// Device/Application/DS6
PROGRAM DS6
VAR
	//massa de dosagem do equipamento em Tonelada.
	MASSA:REAL;
	//Velocidade calculda do Dosador em Hz
	VELOCIDADE:REAL;
	//Espera o fluidizador baixar para o peso minino, pois atingiu o peso maximo
	ESPERA_FLUIDIZADOR_BAIXAR_PESO:BOOL;
	//Liga Dosador manual
	LIGA_DS_MANUAL:BOOL;
	//Liga Dosador automatico
	LIGA_DS_AUTO:BOOL;	
END_VAR

//Dosador 6 - sistema antigo ===============================================
//Formula
//    Passo 1:     massa := (tonelada de dosagem * Percentual de dosagem(sem conversao)  * 10)  
//    Passo 2:    Velocidade := ((massa / (altura * largura * densidade * 60)) + PRST_CONSTANTE_A)/PRST_CONSTANTE_B   	
//	  Inicialmente a Constante a:= 0,045046135
//	  Inicialmente a Constante b:= 0,103503475


//Calculo de velocidade ====================================================

//Calcuulo da massa de dosagem do equipamento 
MASSA := (PRST_VEL_PH1_MANUAL * 10 * PRST_PERC_DOSA_DS06 );

//Calculo da velocidade
VELOCIDADE := ((MASSA/(PRST_ALTURA_DS6*PRST_LARGURA_DS6*PRST_DENSIDADE_DS6*60)) + PRST_CONSTANTE_A_DS6)/PRST_CONSTANTE_B_DS6 ; 

IF BTS_MAPH1 = FALSE THEN
	
	//Comando ==================================================================
	IF BTS_DS6 = TRUE AND AL_GERAL = FALSE THEN
		IF LIGA_DS_MANUAL = TRUE THEN
			LIGA_DS_MANUAL := FALSE;			
		ELSE
			LIGA_DS_MANUAL := TRUE;	
		END_IF		
		BTS_DS6 := FALSE;	
	ELSIF AL_GERAL = TRUE THEN  //delsiga em caso de alarme
		LIGA_DS_MANUAL := FALSE;
		BTS_DS6 := FALSE;	
	END_IF	
	
	//em manual desliga comando do automatico
	LIGA_DS_AUTO := FALSE;
	
ELSE
	
	//Liga dosador 
	IF  AL_GERAL = FALSE THEN
		LIGA_DS_AUTO :=TRUE;
	ELSE
		LIGA_DS_AUTO := FALSE;
	END_IF	
	
	//em auto desliga comando do manual
	LIGA_DS_MANUAL := FALSE;
	
END_IF

//zera velocidade do ph com peso maximo
IF LEITURA_PESO_FLUI1 >= PRST_PESO_MAX_FLUID1 THEN
	ESPERA_FLUIDIZADOR_BAIXAR_PESO := TRUE;
END_IF
	
//ativa velocidade do ph com peso minimo
IF LEITURA_PESO_FLUI1 <= PRST_PESO_MIN_FLUID1 THEN
	ESPERA_FLUIDIZADOR_BAIXAR_PESO := FALSE;
END_IF

IF ESPERA_FLUIDIZADOR_BAIXAR_PESO = FALSE THEN
	//Calculo dosagem kg/h em manual
	PRST_VEL_DS6 := VELOCIDADE;
ELSE
	PRST_VEL_DS6 := 0;
END_IF


//Liga dosador
IF LIGA_DS_AUTO = TRUE OR LIGA_DS_MANUAL = TRUE THEN
	SD_DS6 := TRUE;
ELSE
	SD_DS6 := FALSE;
END_IF

//move velocidade
IF SD_DS6 = TRUE THEN
	VEL_DSA6 :=  PRST_VEL_DS6;
	LEITURA_VEL_DSA6 := PRST_VEL_DS6;
ELSE
	VEL_DSA6 :=0;	
	LEITURA_VEL_DSA6 := 0;
END_IF

END_PROGRAM

// Device/Application/DSA7
PROGRAM DSA7
VAR
	//Tempo de Homogenização em TIME
	TEMPO_DESLIGA_ZERAEVENTO:TON;
	//desliga botao limpa evento
	DESLIGA_BT_LIMPA_EVE:BOOL;
	//Liga Dosador manual
	LIGA_DS_MANUAL:BOOL;
	//Liga Dosador automatico
	LIGA_DS_AUTO:BOOL;
	//Espera o fluidizador baixar para o peso minino, pois atingiu o peso maximo
	ESPERA_FLUIDIZADOR_BAIXAR_PESO:BOOL;
		//Tempo desliga reset totalizador 1
	TMR_RESET_TOTAL1:TON;
	//Tempo desliga reset totalizador 2
	TMR_RESET_TOTAL2:TON;
END_VAR

//POU relacionado aos comandos e alarmes do Dosador Gravimetrico 7 MECHATRON D-5A linha 2


//Controle manual PH 2

//IF BTS_MAPH2 = FALSE THEN
//============================================================================
// comandos manuais 
//============================================================================	
	
//Liga dosador 
IF BTS_DS7 = TRUE AND AL_GERAL = FALSE THEN
	IF LIGA_DS_MANUAL = TRUE THEN
		LIGA_DS_MANUAL := FALSE;
		DS07_HAB := FALSE;
	ELSE
		LIGA_DS_MANUAL :=TRUE;
		DS07_HAB := TRUE;
	END_IF
	BTS_DS7 := FALSE;
END_IF

//desliga em caso de alarme
IF AL_GERAL = TRUE THEN
		LIGA_DS_MANUAL := FALSE;
END_IF

PRST_VEL_DS7 := LEITURA_BASE_SOP_TORRE * (PRST_PERC_DOSA_DS07 / 100);

//============================================================================
// comandos automatico
//============================================================================		
	
//Liga dosador 
IF SD_VLR = TRUE AND SOPRO_SEM_PH = FALSE AND AL_GERAL = FALSE THEN	
	LIGA_DS_AUTO :=TRUE;
	PRST_VEL_DS7 := LEITURA_BASE_SOP_TORRE * (PRST_PERC_DOSA_DS07 / 100);
ELSE
	LIGA_DS_AUTO := FALSE;
	PRST_VEL_DS7 := 0;
END_IF

//Liga dosador
IF LIGA_DS_AUTO = TRUE AND LIGA_DS_MANUAL = TRUE AND AL_GERAL = FALSE THEN
	LIGA_DS7 := TRUE;
	SD_RoscaCelquim := TRUE; 
ELSE
	LIGA_DS7 := FALSE;
	SD_RoscaCelquim := FALSE; 
END_IF


//============================================================================
//  escrita da velocidade
//============================================================================

//Inversão da word da variavel da GVLPH: PRST_VEL_DS7, para variavel da GVLSCHENCK: PESO_DSA7
%QW15080 := %QW12744;
%QW15082 := %QW12742;

//============================================================================
// comandos que independem do comando manual/auto
//============================================================================

//conta tempo de homogenização
TEMPO_DESLIGA_ZERAEVENTO(IN:=BTS_LIMPEVE_DS7,PT:=T#10S);
DESLIGA_BT_LIMPA_EVE := TEMPO_DESLIGA_ZERAEVENTO.Q ;

IF DESLIGA_BT_LIMPA_EVE = TRUE THEN
	BTS_LIMPEVE_DS7 := FALSE;
END_IF

//bits de comando ============================================================
//Os bits de escrita inicio e parada da balança é invertido, por exemplo, para ligar o bit0 = false, e para parar o bit1=false

//Bit iniciar balança
IF LIGA_DS7 = FALSE THEN
	%QX15011.0 := FALSE;    //bit de ligar dosador, false para ativar	
ELSE
	%QX15011.0 := TRUE;		//bit de ligar dosador, true desativa	
END_IF

//bit parar balança
IF LIGA_DS7 = FALSE THEN
	%QX15011.1 := TRUE;		//bit de desligar dosador, true desativar
ELSE		
	%QX15011.1 := FALSE;	//bit de desligar dosador, false ativa	
END_IF

//bit limpar eventos
IF BTS_LIMPEVE_DS7 = TRUE THEN
	%QX15011.2 := TRUE;
ELSE
	%QX15011.2 := FALSE;
END_IF

//bit liberar
%QX15011.3 := TRUE;

//bit modo Volumetrico
IF BTS_MODVOL_DS7 = TRUE THEN
	%QX15011.4 := TRUE;
ELSE
	%QX15011.4 := FALSE;
END_IF
	
//bit modo Gravimetrico
IF BTS_MODGRAV_DS7 = TRUE THEN
	%QX15011.5 := TRUE;
ELSE
	%QX15011.5 := FALSE;
END_IF

//bit reinicializar Totalizador 1
IF BTS_ZERATOTAL1_DS7 = TRUE THEN
	%QX15011.6 := TRUE;
ELSE
	%QX15011.6 := FALSE;
END_IF

//Comando do Reset dos totalizadores geral, apontamento de producao
BTS_ZERATOTAL1_DS7 := BTS_RESET_TOTAL_SCHENCK;
//Tempo desliga reset totalizador 1
TMR_RESET_TOTAL1(IN:= BTS_ZERATOTAL1_DS7, PT:= T#15S);
//desliga o reset do totalizador ao zerar 
IF TMR_RESET_TOTAL1.Q = TRUE THEN
	BTS_ZERATOTAL1_DS7 := FALSE;
	BTS_RESET_TOTAL_SCHENCK := FALSE;
END_IF

//bit reinicializar Totalizador 2
IF BTS_ZERATOTAL2_DS7 = TRUE THEN
	%QX15011.7 := TRUE;
ELSE
	%QX15011.7 := FALSE;
END_IF
//Tempo desliga reset totalizador 2
TMR_RESET_TOTAL2(IN:= BTS_ZERATOTAL2_DS7, PT:= T#15S);
//desliga o reset do totalizador ao zerar 
IF TMR_RESET_TOTAL2.Q = TRUE THEN
	BTS_ZERATOTAL2_DS7 := FALSE;
END_IF


//bit Volume Sincrono
%QX15010.0 := TRUE;

//bit corre. umidade on
%QX15010.1 := TRUE;

//bit corre. umidade off
%QX15010.2 := TRUE;

//bit acionamento med. off
%QX15010.3 := TRUE;

//bit retorno da comporta PMS
%QX15010.4 := TRUE;

//bit reservado
%QX15010.5 := TRUE;

//bit reservado
%QX15010.6 := TRUE;

//bit reservado
%QX15010.7 := TRUE;


//====================================================================================
// Leitura Valores REAL 
//====================================================================================

//Totalizador1, leitura em Kg, 
//Inversão da word da variavel da GVLSCHENCK: LEITURA_TOTALIZADOR1_DSA7, para variavel da GVLPH: TOTALIZADOR1_KG 
%QW10080 := %IW15152;
%QW10082 := %IW15150;

//Totalizador2, leitura em Kg, apenas invertidos as words
//Inversão da word da variavel da GVLSCHENCK: LEITURA_TOTALIZADOR2_DSA7, para variavel da GVLPH: TOTALIZADOR2_KG 
%QW10084 := %IW15212;
%QW10086 := %IW15210;

//Totalizador3, leitura em Tonelada, invertidos as words e dividido por 1000 
//Inversão da word da variavel da GVLSCHENCK: LEITURA_TOTALIZADOR3_DSA7, para variavel da GVLPH: TOTALIZADOR3_KG 
%QW10088 := %IW15322;
%QW10090 := %IW15320;
TOTALIZADOR3_TON_DS7 := TOTALIZADOR3_KG_DS7 / 1000;

//Velocidade atual do dosador
%QW10320 := %IW15272;
%QW10322 := %IW15270;

VELOCIDADE_REAL_DS7 := VELOCIDADE_REAL2_DS7 ;

END_PROGRAM

// Device/Application/DSA8
PROGRAM DSA8
VAR
	//Tempo de Homogenização em TIME
	TEMPO_DESLIGA_ZERAEVENTO:TON;
	//desliga botao limpa evento
	DESLIGA_BT_LIMPA_EVE:BOOL;
	//Liga Dosador manual
	LIGA_DS_MANUAL:BOOL;
	//Liga Dosador automatico
	LIGA_DS_AUTO:BOOL;
	//Espera o fluidizador baixar para o peso minino, pois atingiu o peso maximo
	ESPERA_FLUIDIZADOR_BAIXAR_PESO:BOOL;
	//Tempo desliga reset totalizador 1
	TMR_RESET_TOTAL1:TON;
	//Tempo desliga reset totalizador 2
	TMR_RESET_TOTAL2:TON;
END_VAR

//POU relacionado aos comandos e alarmes do Dosador Gravimetrico 8 MECHATRON D-7A linha 2


//Controle manual PH 2

IF BTS_MAPH2 = FALSE THEN
//============================================================================
// comandos manuais 
//============================================================================	
	
	//Liga dosador 
	IF BTS_DS8 = TRUE AND AL_GERAL = FALSE THEN
		IF LIGA_DS_MANUAL = TRUE THEN
			LIGA_DS_MANUAL := FALSE;
		ELSE
			LIGA_DS_MANUAL :=TRUE;
		END_IF
		BTS_DS8 := FALSE;
	END_IF
	//desliga em caso de alarme
	IF AL_GERAL = TRUE THEN
		LIGA_DS_MANUAL := FALSE;
	END_IF

	//Calculo dosagem kg/h em manual
	PRST_VEL_DS8 := (PRST_VEL_PH2_MANUAL * 1000) * (PRST_PERC_DOSA_DS08 / 100);
	
	//em manual desliga comando do automatico
	LIGA_DS_AUTO := FALSE;	
ELSE
	
//============================================================================
// comandos automatico
//============================================================================		
	
	//Liga dosador 
	IF  AL_GERAL = FALSE THEN
		LIGA_DS_AUTO :=TRUE;
	ELSE
		LIGA_DS_AUTO := FALSE;
	END_IF
	
	//zera velocidade do ph com peso maximo
	IF LEITURA_PESO_FLUI2 >= PRST_PESO_MAX_FLUID2 THEN
		ESPERA_FLUIDIZADOR_BAIXAR_PESO := TRUE;
	END_IF
	
	//ativa velocidade do ph com peso minimo
	IF LEITURA_PESO_FLUI2 <= PRST_PESO_MIN_FLUID2 THEN
		ESPERA_FLUIDIZADOR_BAIXAR_PESO := FALSE;
	END_IF
	
	IF ESPERA_FLUIDIZADOR_BAIXAR_PESO = FALSE THEN
		//Calculo dosagem kg/h em manual
		PRST_VEL_DS8 := (VELOCIDADE_PH2_AUTO) * (PRST_PERC_DOSA_DS08 / 100);
	ELSE
		PRST_VEL_DS8 := 0;
	END_IF
	
	
	//em auto desliga comando do manual
	LIGA_DS_MANUAL := FALSE;
END_IF

//Liga dosador
IF LIGA_DS_AUTO = TRUE OR LIGA_DS_MANUAL = TRUE THEN
	LIGA_DS8 := TRUE;
ELSE
	LIGA_DS8 := FALSE;
END_IF

//============================================================================
//  escrita da velocidade
//============================================================================

//Inversão da word da variavel da GVLPH: PRST_VEL_DS8, para variavel da GVLSCHENCK: PESO_DSA8
%QW15084 := %QW12748;
%QW15086 := %QW12746;

//============================================================================
// comandos que independem do comando manual/auto
//============================================================================

//conta tempo de homogenização
TEMPO_DESLIGA_ZERAEVENTO(IN:=BTS_LIMPEVE_DS8,PT:=T#10S);
DESLIGA_BT_LIMPA_EVE := TEMPO_DESLIGA_ZERAEVENTO.Q ;

IF DESLIGA_BT_LIMPA_EVE = TRUE THEN
	BTS_LIMPEVE_DS8 := FALSE;
END_IF

//bits de comando ============================================================
//Os bits de escrita inicio e parada da balança é invertido, por exemplo, para ligar o bit0 = false, e para parar o bit1=false

//Bit iniciar balança
IF LIGA_DS8 = FALSE THEN
	%QX15013.0 := FALSE;    //bit de ligar dosador, false para ativar	
ELSE
	%QX15013.0 := TRUE;		//bit de ligar dosador, true desativa	
END_IF

//bit parar balança
IF LIGA_DS8 = FALSE THEN
	%QX15013.1 := TRUE;		//bit de desligar dosador, true desativar
ELSE		
	%QX15013.1 := FALSE;	//bit de desligar dosador, false ativa	
END_IF

//bit limpar eventos
IF BTS_LIMPEVE_DS8 = TRUE THEN
	%QX15013.2 := TRUE;
ELSE
	%QX15013.2 := FALSE;
END_IF

//bit liberar
%QX15013.3 := TRUE;

//bit modo Volumetrico
IF BTS_MODVOL_DS8 = TRUE THEN
	%QX15013.4 := TRUE;
ELSE
	%QX15013.4 := FALSE;
END_IF
	
//bit modo Gravimetrico
IF BTS_MODGRAV_DS8 = TRUE THEN
	%QX15013.5 := TRUE;
ELSE
	%QX15013.5 := FALSE;
END_IF

//bit reinicializar Totalizador 1
IF BTS_ZERATOTAL1_DS8 = TRUE THEN
	%QX15013.6 := TRUE;
ELSE
	%QX15013.6 := FALSE;
END_IF

//Comando do Reset dos totalizadores geral, apontamento de producao
BTS_ZERATOTAL1_DS8 := BTS_RESET_TOTAL_SCHENCK;
//Tempo desliga reset totalizador 1
TMR_RESET_TOTAL1(IN:= BTS_ZERATOTAL1_DS8, PT:= T#15S);
//desliga o reset do totalizador ao zerar 
IF TMR_RESET_TOTAL1.Q = TRUE THEN
	BTS_ZERATOTAL1_DS8 := FALSE;
	BTS_RESET_TOTAL_SCHENCK := FALSE;
END_IF

//bit reinicializar Totalizador 2
IF BTS_ZERATOTAL2_DS8 = TRUE THEN
	%QX15013.7 := TRUE;
ELSE
	%QX15013.7 := FALSE;
END_IF
//Tempo desliga reset totalizador 2
TMR_RESET_TOTAL2(IN:= BTS_ZERATOTAL2_DS8, PT:= T#15S);
//desliga o reset do totalizador ao zerar 
IF TMR_RESET_TOTAL2.Q = TRUE THEN
	BTS_ZERATOTAL2_DS8 := FALSE;
END_IF

//bit Volume Sincrono
%QX15012.0 := TRUE;

//bit corre. umidade on
%QX15012.1 := TRUE;

//bit corre. umidade off
%QX15012.2 := TRUE;

//bit acionamento med. off
%QX15012.3 := TRUE;

//bit retorno da comporta PMS
%QX15012.4 := TRUE;

//bit reservado
%QX15012.5 := TRUE;

//bit reservado
%QX15012.6 := TRUE;

//bit reservado
%QX15012.7 := TRUE;


//====================================================================================
// Leitura Valores REAL 
//====================================================================================

//Totalizador1, leitura em Kg, 
//Inversão da word da variavel da GVLSCHENCK: LEITURA_TOTALIZADOR1_DSA8, para variavel da GVLPH: TOTALIZADOR1_KG 
%QW10096 := %IW15156;
%QW10098 := %IW15154;

//Totalizador2, leitura em Kg, apenas invertidos as words
//Inversão da word da variavel da GVLSCHENCK: LEITURA_TOTALIZADOR2_DSA8, para variavel da GVLPH: TOTALIZADOR2_KG 
%QW10100 := %IW15216;
%QW10102 := %IW15214;

//Totalizador3, leitura em Tonelada, invertidos as words e dividido por 1000 
//Inversão da word da variavel da GVLSCHENCK: LEITURA_TOTALIZADOR3_DSA8, para variavel da GVLPH: TOTALIZADOR3_KG 
%QW10104 := %IW15326;
%QW10106 := %IW15324;
TOTALIZADOR3_TON_DS8 := TOTALIZADOR3_KG_DS8 / 1000;

//Velocidade atual do dosador
%QW10324 := %IW15276;
%QW10326 := %IW15274;

VELOCIDADE_REAL_DS8 := VELOCIDADE_REAL2_DS8 ;

END_PROGRAM

// Device/Application/DSA9
PROGRAM DSA9
VAR
	//Tempo de Homogenização em TIME
	TEMPO_DESLIGA_ZERAEVENTO:TON;
	//desliga botao limpa evento
	DESLIGA_BT_LIMPA_EVE:BOOL;
	//Liga Dosador manual
	LIGA_DS_MANUAL:BOOL;
	//Liga Dosador automatico
	LIGA_DS_AUTO:BOOL;
	//Espera o fluidizador baixar para o peso minino, pois atingiu o peso maximo
	ESPERA_FLUIDIZADOR_BAIXAR_PESO:BOOL;
	//Tempo desliga reset totalizador 1
	TMR_RESET_TOTAL1:TON;
	//Tempo desliga reset totalizador 2
	TMR_RESET_TOTAL2:TON;

END_VAR

//POU relacionado aos comandos e alarmes do Dosador Gravimetrico 9 MECHATRON D-6A linha 2	


//Controle manual PH 2

IF BTS_MAPH2 = FALSE THEN
//============================================================================
// comandos manuais 
//============================================================================	
	
	//Liga dosador 
	IF BTS_DS9 = TRUE AND AL_GERAL = FALSE THEN
		IF LIGA_DS_MANUAL = TRUE THEN
			LIGA_DS_MANUAL := FALSE;
		ELSE
			LIGA_DS_MANUAL :=TRUE;
		END_IF
		BTS_DS9 := FALSE;
	END_IF
	//desliga em caso de alarme
	IF AL_GERAL = TRUE THEN
		LIGA_DS_MANUAL := FALSE;
	END_IF
	
	//Calculo dosagem kg/h em manual
	PRST_VEL_DS9 := (PRST_VEL_PH2_MANUAL * 1000) * (PRST_PERC_DOSA_DS09 / 100);

	//em manual desliga comando do automatico
	LIGA_DS_AUTO := FALSE;
	
ELSE
	
//============================================================================
// comandos automatico
//============================================================================		
	
	//Liga dosador 
	IF  AL_GERAL = FALSE THEN
		LIGA_DS_AUTO :=TRUE;
	ELSE
		LIGA_DS_AUTO := FALSE;
	END_IF
	
	//zera velocidade do ph com peso maximo
	IF LEITURA_PESO_FLUI2 >= PRST_PESO_MAX_FLUID2 THEN
		ESPERA_FLUIDIZADOR_BAIXAR_PESO := TRUE;
	END_IF
	
	//ativa velocidade do ph com peso minimo
	IF LEITURA_PESO_FLUI2 <= PRST_PESO_MIN_FLUID2 THEN
		ESPERA_FLUIDIZADOR_BAIXAR_PESO := FALSE;
	END_IF
	
	IF ESPERA_FLUIDIZADOR_BAIXAR_PESO = FALSE THEN
		//Calculo dosagem kg/h em manual
		PRST_VEL_DS9 := (VELOCIDADE_PH2_AUTO) * (PRST_PERC_DOSA_DS09 / 100);
	ELSE
		PRST_VEL_DS9 := 0;	
	END_IF
	
	
	//em auto desliga comando do manual
	LIGA_DS_MANUAL := FALSE;
END_IF

//Liga dosador
IF LIGA_DS_AUTO = TRUE OR LIGA_DS_MANUAL = TRUE THEN
	LIGA_DS9 := TRUE;
ELSE
	LIGA_DS9 := FALSE;
END_IF

//============================================================================
//  escrita da velocidade
//============================================================================

//Inversão da word da variavel da GVLPH: PRST_VEL_DS9, para variavel da GVLSCHENCK: PESO_DSA9
%QW15088 := %QW12752;
%QW15090 := %QW12750;


//============================================================================
// comandos que independem do comando manual/auto
//============================================================================

//conta tempo de homogenização
TEMPO_DESLIGA_ZERAEVENTO(IN:=BTS_LIMPEVE_DS9,PT:=T#10S);
DESLIGA_BT_LIMPA_EVE := TEMPO_DESLIGA_ZERAEVENTO.Q ;

IF DESLIGA_BT_LIMPA_EVE = TRUE THEN
	BTS_LIMPEVE_DS9 := FALSE;
END_IF

//bits de comando ============================================================
//Os bits de escrita inicio e parada da balança é invertido, por exemplo, para ligar o bit0 = false, e para parar o bit1=false

//Bit iniciar balança
IF LIGA_DS9 = FALSE THEN
	%QX15015.0 := FALSE;    //bit de ligar dosador, false para ativar	
ELSE
	%QX15015.0 := TRUE;		//bit de ligar dosador, true desativa	
END_IF

//bit parar balança
IF LIGA_DS9 = FALSE THEN
	%QX15015.1 := TRUE;		//bit de desligar dosador, true desativar
ELSE		
	%QX15015.1 := FALSE;	//bit de desligar dosador, false ativa	
END_IF

//bit limpar eventos
IF BTS_LIMPEVE_DS9 = TRUE THEN
	%QX15015.2 := TRUE;
ELSE
	%QX15015.2 := FALSE;
END_IF

//bit liberar
%QX15015.3 := TRUE;

//bit modo Volumetrico
IF BTS_MODVOL_DS9 = TRUE THEN
	%QX15015.4 := TRUE;
ELSE
	%QX15015.4 := FALSE;
END_IF
	
//bit modo Gravimetrico
IF BTS_MODGRAV_DS9 = TRUE THEN
	%QX15015.5 := TRUE;
ELSE
	%QX15015.5 := FALSE;
END_IF

//bit reinicializar Totalizador 1
IF BTS_ZERATOTAL1_DS9 = TRUE THEN
	%QX15015.6 := TRUE;
ELSE
	%QX15015.6 := FALSE;
END_IF

//Comando do Reset dos totalizadores geral, apontamento de producao
BTS_ZERATOTAL1_DS9 := BTS_RESET_TOTAL_SCHENCK;
//Tempo desliga reset totalizador 1
TMR_RESET_TOTAL1(IN:= BTS_ZERATOTAL1_DS9, PT:= T#15S);
//desliga o reset do totalizador ao zerar 
IF TMR_RESET_TOTAL1.Q = TRUE THEN
	BTS_ZERATOTAL1_DS9 := FALSE;
	BTS_RESET_TOTAL_SCHENCK := FALSE;
END_IF

//bit reinicializar Totalizador 2
IF BTS_ZERATOTAL2_DS9 = TRUE THEN
	%QX15015.7 := TRUE;
ELSE
	%QX15015.7 := FALSE;
END_IF
//Tempo desliga reset totalizador 2
TMR_RESET_TOTAL2(IN:= BTS_ZERATOTAL2_DS9, PT:= T#15S);
//desliga o reset do totalizador ao zerar 
IF TMR_RESET_TOTAL2.Q = TRUE THEN
	BTS_ZERATOTAL2_DS9 := FALSE;
END_IF

//bit Volume Sincrono
%QX15014.0 := TRUE;

//bit corre. umidade on
%QX15014.1 := TRUE;

//bit corre. umidade off
%QX15014.2 := TRUE;

//bit acionamento med. off
%QX15014.3 := TRUE;

//bit retorno da comporta PMS
%QX15014.4 := TRUE;

//bit reservado
%QX15014.5 := TRUE;

//bit reservado
%QX15014.6 := TRUE;

//bit reservado
%QX15014.7 := TRUE;


//====================================================================================
// Leitura Valores REAL 
//====================================================================================

//Totalizador1, leitura em Kg, 
//Inversão da word da variavel da GVLSCHENCK: LEITURA_TOTALIZADOR1_DSA9, para variavel da GVLPH: TOTALIZADOR1_KG 
%QW10112 := %IW15160;
%QW10114 := %IW15158;

//Totalizador2, leitura em Kg, apenas invertidos as words
//Inversão da word da variavel da GVLSCHENCK: LEITURA_TOTALIZADOR2_DSA9, para variavel da GVLPH: TOTALIZADOR2_KG 
%QW10116 := %IW15220;
%QW10118 := %IW15218;

//Totalizador3, leitura em Tonelada, invertidos as words e dividido por 1000 
//Inversão da word da variavel da GVLSCHENCK: LEITURA_TOTALIZADOR3_DSA9, para variavel da GVLPH: TOTALIZADOR3_KG 
%QW10120 := %IW15330;
%QW10122 := %IW15328;
TOTALIZADOR3_TON_DS9 := TOTALIZADOR3_KG_DS9 / 1000;

//Velocidade atual do dosador
%QW10328 := %IW15280;
%QW10330 := %IW15278;

VELOCIDADE_REAL_DS9 := VELOCIDADE_REAL2_DS9;

END_PROGRAM

// Device/Application/DSA10
PROGRAM DSA10
VAR
	//Tempo de Homogenização em TIME
	TEMPO_DESLIGA_ZERAEVENTO:TON;
	//desliga botao limpa evento
	DESLIGA_BT_LIMPA_EVE:BOOL;
	//Liga Dosador manual
	LIGA_DS_MANUAL:BOOL;
	//Liga Dosador automatico
	LIGA_DS_AUTO:BOOL;
	//Espera o fluidizador baixar para o peso minino, pois atingiu o peso maximo
	ESPERA_FLUIDIZADOR_BAIXAR_PESO:BOOL;
	//Tempo desliga reset totalizador 1
	TMR_RESET_TOTAL1:TON;
	//Tempo desliga reset totalizador 2
	TMR_RESET_TOTAL2:TON;
END_VAR

//POU relacionado aos comandos e alarmes do Dosador Gravimetrico 10 MECHATRON DEA-4A linha 2	


//Controle manual PH 2

IF BTS_MAPH2 = FALSE THEN
//============================================================================
// comandos manuais 
//============================================================================	
	
	//Liga dosador 
	IF BTS_DS10 = TRUE AND AL_GERAL = FALSE THEN
		IF LIGA_DS_MANUAL = TRUE THEN
			LIGA_DS_MANUAL := FALSE;
		ELSE
			LIGA_DS_MANUAL :=TRUE;
		END_IF
		BTS_DS10 := FALSE;
	END_IF
	//desliga em caso de alarme
	IF AL_GERAL = TRUE THEN
		LIGA_DS_MANUAL := FALSE;
	END_IF

	//Calculo dosagem kg/h em manual
	PRST_VEL_DS10 := (PRST_VEL_PH2_MANUAL * 1000) * (PRST_PERC_DOSA_DS10 / 100);
	
	
	//em manual desliga comando do automatico
	LIGA_DS_AUTO := FALSE;
	
ELSE
//============================================================================
// comandos automatico
//============================================================================		
	
	//Liga dosador 
	IF  AL_GERAL = FALSE THEN
		LIGA_DS_AUTO :=TRUE;
	ELSE
		LIGA_DS_AUTO := FALSE;
	END_IF
	
	
	//zera velocidade do ph com peso maximo
	IF LEITURA_PESO_FLUI2 >= PRST_PESO_MAX_FLUID2 THEN
		ESPERA_FLUIDIZADOR_BAIXAR_PESO := TRUE;
	END_IF
	
	//ativa velocidade do ph com peso minimo
	IF LEITURA_PESO_FLUI2 <= PRST_PESO_MIN_FLUID2 THEN
		ESPERA_FLUIDIZADOR_BAIXAR_PESO := FALSE;
	END_IF
	
	IF ESPERA_FLUIDIZADOR_BAIXAR_PESO = FALSE THEN
		//Calculo dosagem kg/h em manual
		PRST_VEL_DS10 := (VELOCIDADE_PH2_AUTO) * (PRST_PERC_DOSA_DS10 / 100);
	ELSE
		PRST_VEL_DS10 := 0;
	END_IF
	
	//em auto desliga comando do manual
	LIGA_DS_MANUAL := FALSE;
	
END_IF

//Liga dosador
IF LIGA_DS_AUTO = TRUE OR LIGA_DS_MANUAL = TRUE THEN
	LIGA_DS10 := TRUE;
ELSE
	LIGA_DS10 := FALSE;
END_IF

//============================================================================
//  escrita da velocidade
//============================================================================

//Inversão da word da variavel da GVLPH: PRST_VEL_DS10, para variavel da GVLSCHENCK: PESO_DSA10
%QW15092 := %QW12756;
%QW15094 := %QW12754;

//============================================================================
// comandos que independem do comando manual/auto
//============================================================================

//conta tempo de homogenização
TEMPO_DESLIGA_ZERAEVENTO(IN:=BTS_LIMPEVE_DS10,PT:=T#10S);
DESLIGA_BT_LIMPA_EVE := TEMPO_DESLIGA_ZERAEVENTO.Q ;

IF DESLIGA_BT_LIMPA_EVE = TRUE THEN
	BTS_LIMPEVE_DS10 := FALSE;
END_IF

//bits de comando ============================================================
//Os bits de escrita inicio e parada da balança é invertido, por exemplo, para ligar o bit0 = false, e para parar o bit1=false

//Bit iniciar balança
IF LIGA_DS10 = FALSE THEN
	%QX15017.0 := FALSE;    //bit de ligar dosador, false para ativar	
ELSE
	%QX15017.0 := TRUE;		//bit de ligar dosador, true desativa	
END_IF

//bit parar balança
IF LIGA_DS10 = FALSE THEN
	%QX15017.1 := TRUE;		//bit de desligar dosador, true desativar
ELSE		
	%QX15017.1 := FALSE;	//bit de desligar dosador, false ativa	
END_IF

//bit limpar eventos
IF BTS_LIMPEVE_DS10 = TRUE THEN
	%QX15017.2 := TRUE;
ELSE
	%QX15017.2 := FALSE;
END_IF

//bit liberar
%QX15017.3 := TRUE;

//bit modo Volumetrico
IF BTS_MODVOL_DS10 = TRUE THEN
	%QX15017.4 := TRUE;
ELSE
	%QX15017.4 := FALSE;
END_IF
	
//bit modo Gravimetrico
IF BTS_MODGRAV_DS10 = TRUE THEN
	%QX15017.5 := TRUE;
ELSE
	%QX15017.5 := FALSE;
END_IF

//bit reinicializar Totalizador 1
IF BTS_ZERATOTAL1_DS10 = TRUE THEN
	%QX15017.6 := TRUE;
ELSE
	%QX15017.6 := FALSE;
END_IF

//Comando do Reset dos totalizadores geral, apontamento de producao
BTS_ZERATOTAL1_DS10 := BTS_RESET_TOTAL_SCHENCK;
//Tempo desliga reset totalizador 1
TMR_RESET_TOTAL1(IN:= BTS_ZERATOTAL1_DS10, PT:= T#15S);
//desliga o reset do totalizador ao zerar 
IF TMR_RESET_TOTAL1.Q = TRUE THEN
	BTS_ZERATOTAL1_DS10 := FALSE;
	BTS_RESET_TOTAL_SCHENCK := FALSE;
END_IF

//bit reinicializar Totalizador 2
IF BTS_ZERATOTAL2_DS10 = TRUE THEN
	%QX15017.7 := TRUE;
ELSE
	%QX15017.7 := FALSE;
END_IF
//Tempo desliga reset totalizador 2
TMR_RESET_TOTAL2(IN:= BTS_ZERATOTAL2_DS10, PT:= T#15S);
//desliga o reset do totalizador ao zerar 
IF TMR_RESET_TOTAL2.Q = TRUE THEN
	BTS_ZERATOTAL2_DS10 := FALSE;
END_IF

//bit Volume Sincrono
%QX15016.0 := TRUE;

//bit corre. umidade on
%QX15016.1 := TRUE;

//bit corre. umidade off
%QX15016.2 := TRUE;

//bit acionamento med. off
%QX15016.3 := TRUE;

//bit retorno da comporta PMS
%QX15016.4 := TRUE;

//bit reservado
%QX15016.5 := TRUE;

//bit reservado
%QX15016.6 := TRUE;

//bit reservado
%QX15016.7 := TRUE;


//====================================================================================
// Leitura Valores REAL 
//====================================================================================

//Totalizador1, leitura em Kg, 
//Inversão da word da variavel da GVLSCHENCK: LEITURA_TOTALIZADOR1_DSA10, para variavel da GVLPH: TOTALIZADOR1_KG 
%QW10128 := %IW15164;
%QW10130 := %IW15162;

//Totalizador2, leitura em Kg, apenas invertidos as words
//Inversão da word da variavel da GVLSCHENCK: LEITURA_TOTALIZADOR2_DSA10, para variavel da GVLPH: TOTALIZADOR2_KG 
%QW10132 := %IW15224;
%QW10134 := %IW15222;

//Totalizador3, leitura em Tonelada, invertidos as words e dividido por 1000 
//Inversão da word da variavel da GVLSCHENCK: LEITURA_TOTALIZADOR3_DSA10, para variavel da GVLPH: TOTALIZADOR3_KG 
%QW10136 := %IW15334;
%QW10138 := %IW15332;
TOTALIZADOR3_TON_DS10 := TOTALIZADOR3_KG_DS10 / 1000;

//Velocidade atual do dosador
%QW10332 := %IW15284;
%QW10334 := %IW15282;

VELOCIDADE_REAL_DS10 := VELOCIDADE_REAL2_DS10;

END_PROGRAM

// Device/Application/DSA11
PROGRAM DSA11
VAR
	//Tempo de Homogenização em TIME
	TEMPO_DESLIGA_ZERAEVENTO:TON;
	//desliga botao limpa evento
	DESLIGA_BT_LIMPA_EVE:BOOL;
	//Liga Dosador manual
	LIGA_DS_MANUAL:BOOL;
	//Liga Dosador automatico
	LIGA_DS_AUTO:BOOL; 
	//Espera o fluidizador baixar para o peso minino, pois atingiu o peso maximo
	ESPERA_FLUIDIZADOR_BAIXAR_PESO:BOOL;
	//Tempo desliga reset totalizador 1
	TMR_RESET_TOTAL1:TON;
	//Tempo desliga reset totalizador 2
	TMR_RESET_TOTAL2:TON;
END_VAR

//POU relacionado aos comandos e alarmes do Dosador Gravimetrico 11 MECHATRON DEA-2A linha 2 - Po Base 11


//Controle manual PH 2

IF BTS_MAPH2 = FALSE THEN
//============================================================================
// comandos manuais 
//============================================================================	
	
	//Liga dosador 
	IF BTS_DS11 = TRUE AND AL_GERAL = FALSE THEN
		IF LIGA_DS_MANUAL = TRUE THEN
			LIGA_DS_MANUAL := FALSE;
		ELSE
			LIGA_DS_MANUAL :=TRUE;
		END_IF
		BTS_DS11 := FALSE;
	END_IF
	//desliga em caso de alarme
	IF AL_GERAL = TRUE THEN
		LIGA_DS_MANUAL := FALSE;
	END_IF
	
	//Calculo dosagem kg/h em manual
	PRST_VEL_DS11 := (PRST_VEL_PH2_MANUAL * 1000) * (PRST_PERC_DOSA_PB11 / 100);		
	
	//em manual desliga comando do automatico
	LIGA_DS_AUTO := FALSE;
	
ELSE
//============================================================================
// comandos automatico
//============================================================================		
	
	//Liga dosador 
	IF  AL_GERAL = FALSE THEN
		LIGA_DS_AUTO :=TRUE;
	ELSE
		LIGA_DS_AUTO := FALSE;
	END_IF
	
	//zera velocidade do ph com peso maximo
	IF LEITURA_PESO_FLUI2 >= PRST_PESO_MAX_FLUID2 THEN
		ESPERA_FLUIDIZADOR_BAIXAR_PESO := TRUE;
	END_IF
	
	//ativa velocidade do ph com peso minimo
	IF LEITURA_PESO_FLUI2 <= PRST_PESO_MIN_FLUID2 THEN
		ESPERA_FLUIDIZADOR_BAIXAR_PESO := FALSE;
	END_IF

	IF ESPERA_FLUIDIZADOR_BAIXAR_PESO = FALSE THEN
		//Calculo dosagem kg/h em manual
		PRST_VEL_DS11 := (VELOCIDADE_PH2_AUTO) * (PRST_PERC_DOSA_PB11 / 100);
	ELSE
		PRST_VEL_DS11 := 0;
	END_IF
	
	
	//em auto desliga comando do manual
	LIGA_DS_MANUAL := FALSE;
	
END_IF

//Liga dosador
IF LIGA_DS_AUTO = TRUE OR LIGA_DS_MANUAL = TRUE THEN
	LIGA_DS11 := TRUE;
ELSE
	LIGA_DS11 := FALSE;
END_IF


//============================================================================
//  escrita da velocidade
//============================================================================

//Inversão da word da variavel da GVLPH: PRST_VEL_DS11, para variavel da GVLSCHENCK: PESO_DSA11
%QW15096 := %QW12760;
%QW15098 := %QW12758;

//============================================================================
// comandos que independem do comando manual/auto
//============================================================================

//conta tempo de homogenização
TEMPO_DESLIGA_ZERAEVENTO(IN:=BTS_LIMPEVE_DS11,PT:=T#10S);
DESLIGA_BT_LIMPA_EVE := TEMPO_DESLIGA_ZERAEVENTO.Q ;

IF DESLIGA_BT_LIMPA_EVE = TRUE THEN
	BTS_LIMPEVE_DS11 := FALSE;
END_IF

//bits de comando ============================================================
//Os bits de escrita inicio e parada da balança é invertido, por exemplo, para ligar o bit0 = false, e para parar o bit1=false

//Bit iniciar balança
IF LIGA_DS11 = FALSE THEN
	%QX15019.0 := FALSE;    //bit de ligar dosador, false para ativar	
ELSE
	%QX15019.0 := TRUE;		//bit de ligar dosador, true desativa	
END_IF

//bit parar balança
IF LIGA_DS11 = FALSE THEN
	%QX15019.1 := TRUE;		//bit de desligar dosador, true desativar
ELSE		
	%QX15019.1 := FALSE;	//bit de desligar dosador, false ativa	
END_IF

//bit limpar eventos
IF BTS_LIMPEVE_DS11 = TRUE THEN
	%QX15019.2 := TRUE;
ELSE
	%QX15019.2 := FALSE;
END_IF

//bit liberar
%QX15019.3 := TRUE;

//bit modo Volumetrico
IF BTS_MODVOL_DS11 = TRUE THEN
	%QX15019.4 := TRUE;
ELSE
	%QX15019.4 := FALSE;
END_IF
	
//bit modo Gravimetrico
IF BTS_MODGRAV_DS11 = TRUE THEN
	%QX15019.5 := TRUE;
ELSE
	%QX15019.5 := FALSE;
END_IF

//bit reinicializar Totalizador 1
IF BTS_ZERATOTAL1_DS11 = TRUE THEN
	%QX15019.6 := TRUE;
ELSE
	%QX15019.6 := FALSE;
END_IF

//Comando do Reset dos totalizadores geral, apontamento de producao
BTS_ZERATOTAL1_DS11 := BTS_RESET_TOTAL_SCHENCK;
//Tempo desliga reset totalizador 1
TMR_RESET_TOTAL1(IN:= BTS_ZERATOTAL1_DS11, PT:= T#15S);
//desliga o reset do totalizador ao zerar 
IF TMR_RESET_TOTAL1.Q = TRUE THEN
	BTS_ZERATOTAL1_DS11 := FALSE;
	BTS_RESET_TOTAL_SCHENCK := FALSE;
END_IF

//bit reinicializar Totalizador 2
IF BTS_ZERATOTAL2_DS11 = TRUE THEN
	%QX15019.7 := TRUE;
ELSE
	%QX15019.7 := FALSE;
END_IF
//Tempo desliga reset totalizador 2
TMR_RESET_TOTAL2(IN:= BTS_ZERATOTAL2_DS11, PT:= T#15S);
//desliga o reset do totalizador ao zerar 
IF TMR_RESET_TOTAL2.Q = TRUE THEN
	BTS_ZERATOTAL2_DS11 := FALSE;
END_IF

//bit Volume Sincrono
%QX15018.0 := TRUE;

//bit corre. umidade on
%QX15018.1 := TRUE;

//bit corre. umidade off
%QX15018.2 := TRUE;

//bit acionamento med. off
%QX15018.3 := TRUE;

//bit retorno da comporta PMS
%QX15018.4 := TRUE;

//bit reservado
%QX15018.5 := TRUE;

//bit reservado
%QX15018.6 := TRUE;

//bit reservado
%QX15018.7 := TRUE;


//====================================================================================
// Leitura Valores REAL 
//====================================================================================

//Totalizador1, leitura em Kg, 
//Inversão da word da variavel da GVLSCHENCK: LEITURA_TOTALIZADOR1_DSA11, para variavel da GVLPH: TOTALIZADOR1_KG 
%QW10144 := %IW15168;
%QW10146 := %IW15166;

//Totalizador2, leitura em Kg, apenas invertidos as words
//Inversão da word da variavel da GVLSCHENCK: LEITURA_TOTALIZADOR2_DSA11, para variavel da GVLPH: TOTALIZADOR2_KG 
%QW10148 := %IW15228;
%QW10150 := %IW15226;

//Totalizador3, leitura em Tonelada, invertidos as words e dividido por 1000 
//Inversão da word da variavel da GVLSCHENCK: LEITURA_TOTALIZADOR3_DSA11, para variavel da GVLPH: TOTALIZADOR3_KG 
%QW10152 := %IW15338;
%QW10154 := %IW15336;
TOTALIZADOR3_TON_DS11 := TOTALIZADOR3_KG_DS11 / 1000;

//Velocidade atual do dosador
%QW10336 := %IW15288;
%QW10338 := %IW15286;

VELOCIDADE_REAL_DS11 := VELOCIDADE_REAL2_DS11;

END_PROGRAM

// Device/Application/DSA12
PROGRAM DSA12
VAR
	//Tempo de Homogenização em TIME
	TEMPO_DESLIGA_ZERAEVENTO:TON;
	//desliga botao limpa evento
	DESLIGA_BT_LIMPA_EVE:BOOL;
	//Liga Dosador manual
	LIGA_DS_MANUAL:BOOL;
	//Liga Dosador automatico
	LIGA_DS_AUTO:BOOL;
	//Espera o fluidizador baixar para o peso minino, pois atingiu o peso maximo
	ESPERA_FLUIDIZADOR_BAIXAR_PESO:BOOL;
	//Tempo desliga reset totalizador 1
	TMR_RESET_TOTAL1:TON;
	//Tempo desliga reset totalizador 2
	TMR_RESET_TOTAL2:TON;
END_VAR

//POU relacionado aos comandos e alarmes do Dosador Gravimetrico 12 MECHATRON DEA-3A linha 2	


//Controle manual PH 2

IF BTS_MAPH2 = FALSE THEN
//============================================================================
// comandos manuais 
//============================================================================	
	
	//Liga dosador 
	IF BTS_DS12 = TRUE AND AL_GERAL = FALSE THEN
		IF LIGA_DS_MANUAL = TRUE THEN
			LIGA_DS_MANUAL := FALSE;
		ELSE
			LIGA_DS_MANUAL :=TRUE;
		END_IF
		BTS_DS12 := FALSE;
	END_IF
	//desliga em caso de alarme
	IF AL_GERAL = TRUE THEN
		LIGA_DS_MANUAL := FALSE;
	END_IF

	//Calculo dosagem kg/h em manual
	PRST_VEL_DS12 := (PRST_VEL_PH2_MANUAL * 1000) * (PRST_PERC_DOSA_DS12 / 100);
	
	//em manual desliga comando do automatico
	LIGA_DS_AUTO := FALSE;	
ELSE
//============================================================================
// comandos automatico
//============================================================================		
	
	//Liga dosador 
	IF  AL_GERAL = FALSE THEN
		LIGA_DS_AUTO :=TRUE;
	ELSE
		LIGA_DS_AUTO := FALSE;
	END_IF
	
	//zera velocidade do ph com peso maximo
	IF LEITURA_PESO_FLUI2 >= PRST_PESO_MAX_FLUID2 THEN
		ESPERA_FLUIDIZADOR_BAIXAR_PESO := TRUE;
	END_IF
	
	//ativa velocidade do ph com peso minimo
	IF LEITURA_PESO_FLUI2 <= PRST_PESO_MIN_FLUID2 THEN
		ESPERA_FLUIDIZADOR_BAIXAR_PESO := FALSE;
	END_IF
	
	IF ESPERA_FLUIDIZADOR_BAIXAR_PESO = FALSE THEN
		//Calculo dosagem kg/h em manual
		PRST_VEL_DS12 := (VELOCIDADE_PH2_AUTO) * (PRST_PERC_DOSA_DS12 / 100);
	ELSE
		PRST_VEL_DS12 := 0;
	END_IF
	
	//em auto desliga comando do manual
	LIGA_DS_MANUAL := FALSE;
	
END_IF

//Liga dosador
IF LIGA_DS_AUTO = TRUE OR LIGA_DS_MANUAL = TRUE THEN
	LIGA_DS12 := TRUE;
ELSE
	LIGA_DS12 := FALSE;
END_IF

//============================================================================
//  escrita da velocidade
//============================================================================

//Inversão da word da variavel da GVLPH: PRST_VEL_DS12, para variavel da GVLSCHENCK: PESO_DSA12
%QW15100 := %QW12764;
%QW15102 := %QW12762;

//============================================================================
// comandos que independem do comando manual/auto
//============================================================================

//conta tempo de homogenização
TEMPO_DESLIGA_ZERAEVENTO(IN:=BTS_LIMPEVE_DS12,PT:=T#10S);
DESLIGA_BT_LIMPA_EVE := TEMPO_DESLIGA_ZERAEVENTO.Q ;

IF DESLIGA_BT_LIMPA_EVE = TRUE THEN
	BTS_LIMPEVE_DS12 := FALSE;
END_IF

//bits de comando ============================================================
//Os bits de escrita inicio e parada da balança é invertido, por exemplo, para ligar o bit0 = false, e para parar o bit1=false

//Bit iniciar balança
IF LIGA_DS12 = FALSE THEN
	%QX15021.0 := FALSE;    //bit de ligar dosador, false para ativar	
ELSE
	%QX15021.0 := TRUE;		//bit de ligar dosador, true desativa	
END_IF

//bit parar balança
IF LIGA_DS12 = FALSE THEN
	%QX15021.1 := TRUE;		//bit de desligar dosador, true desativar
ELSE		
	%QX15021.1 := FALSE;	//bit de desligar dosador, false ativa	
END_IF

//bit limpar eventos
IF BTS_LIMPEVE_DS12 = TRUE THEN
	%QX15021.2 := TRUE;
ELSE
	%QX15021.2 := FALSE;
END_IF

//bit liberar
%QX15021.3 := TRUE;

//bit modo Volumetrico
IF BTS_MODVOL_DS12 = TRUE THEN
	%QX15021.4 := TRUE;
ELSE
	%QX15021.4 := FALSE;
END_IF
	
//bit modo Gravimetrico
IF BTS_MODGRAV_DS12 = TRUE THEN
	%QX15021.5 := TRUE;
ELSE
	%QX15021.5 := FALSE;
END_IF

//bit reinicializar Totalizador 1
IF BTS_ZERATOTAL1_DS12 = TRUE THEN
	%QX15021.6 := TRUE;
ELSE
	%QX15021.6 := FALSE;
END_IF

//Comando do Reset dos totalizadores geral, apontamento de producao
BTS_ZERATOTAL1_DS12 := BTS_RESET_TOTAL_SCHENCK;
//Tempo desliga reset totalizador 1
TMR_RESET_TOTAL1(IN:= BTS_ZERATOTAL1_DS12, PT:= T#15S);
//desliga o reset do totalizador ao zerar 
IF TMR_RESET_TOTAL1.Q = TRUE THEN
	BTS_ZERATOTAL1_DS12 := FALSE;
	BTS_RESET_TOTAL_SCHENCK := FALSE;
END_IF

//bit reinicializar Totalizador 2
IF BTS_ZERATOTAL2_DS12 = TRUE THEN
	%QX15021.7 := TRUE;
ELSE
	%QX15021.7 := FALSE;
END_IF
//Tempo desliga reset totalizador 2
TMR_RESET_TOTAL2(IN:= BTS_ZERATOTAL2_DS12, PT:= T#15S);
//desliga o reset do totalizador ao zerar 
IF TMR_RESET_TOTAL2.Q = TRUE THEN
	BTS_ZERATOTAL2_DS12 := FALSE;
END_IF

//bit Volume Sincrono
%QX15020.0 := TRUE;

//bit corre. umidade on
%QX15020.1 := TRUE;

//bit corre. umidade off
%QX15020.2 := TRUE;

//bit acionamento med. off
%QX15020.3 := TRUE;

//bit retorno da comporta PMS
%QX15020.4 := TRUE;

//bit reservado
%QX15020.5 := TRUE;

//bit reservado
%QX15020.6 := TRUE;

//bit reservado
%QX15020.7 := TRUE;


//====================================================================================
// Leitura Valores REAL 
//====================================================================================

//Totalizador1, leitura em Kg, 
//Inversão da word da variavel da GVLSCHENCK: LEITURA_TOTALIZADOR1_DSA12, para variavel da GVLPH: TOTALIZADOR1_KG 
%QW10160 := %IW15172;
%QW10162 := %IW15170;

//Totalizador2, leitura em Kg, apenas invertidos as words
//Inversão da word da variavel da GVLSCHENCK: LEITURA_TOTALIZADOR2_DSA12, para variavel da GVLPH: TOTALIZADOR2_KG 
%QW10164 := %IW15232;
%QW10166 := %IW15230;

//Totalizador3, leitura em Tonelada, invertidos as words e dividido por 1000 
//Inversão da word da variavel da GVLSCHENCK: LEITURA_TOTALIZADOR3_DSA12, para variavel da GVLPH: TOTALIZADOR3_KG 
%QW10168 := %IW15342;
%QW10170 := %IW15340;
TOTALIZADOR3_TON_DS12 := TOTALIZADOR3_KG_DS12 / 1000;

//Velocidade atual do dosador
%QW10340 := %IW15292;
%QW10342 := %IW15290;

VELOCIDADE_REAL_DS12 := VELOCIDADE_REAL2_DS12;

END_PROGRAM

// Device/Application/DSA14
PROGRAM DSA14
VAR
	//Tempo de Homogenização em TIME
	TEMPO_DESLIGA_ZERAEVENTO:TON;
	//desliga botao limpa evento
	DESLIGA_BT_LIMPA_EVE:BOOL;
	//Liga Dosador manual
	LIGA_DS_MANUAL:BOOL;
	//Liga Dosador automatico
	LIGA_DS_AUTO:BOOL;
	//Espera o fluidizador baixar para o peso minino, pois atingiu o peso maximo
	ESPERA_FLUIDIZADOR_BAIXAR_PESO:BOOL;
	//Tempo desliga reset totalizador 1
	TMR_RESET_TOTAL1:TON;
	//Tempo desliga reset totalizador 2
	TMR_RESET_TOTAL2:TON;
	teste1: WORD;
	teste2: WORD;
	teste3: DWORD;
END_VAR

//POU relacionado aos comandos e alarmes do Dosador Gravimetrico 14 MECHATRON DEA-3A linha 2	


//Controle manual PH 2

IF BTS_MAPH2 = FALSE THEN
//============================================================================
// comandos manuais 
//============================================================================	
	
	//Liga dosador 
	IF BTS_DS14 = TRUE AND AL_GERAL = FALSE THEN
		IF LIGA_DS_MANUAL = TRUE THEN
			LIGA_DS_MANUAL := FALSE;
		ELSE
			LIGA_DS_MANUAL :=TRUE;
		END_IF
		BTS_DS14 := FALSE;
	END_IF
	//desliga em caso de alarme
	IF AL_GERAL = TRUE THEN
		LIGA_DS_MANUAL := FALSE;
	END_IF

	//Calculo dosagem kg/h em manual
	PRST_VEL_DS14 := (PRST_VEL_PH2_MANUAL * 1000) * (PRST_PERC_DOSA_DS14 / 100);
	
	//em manual desliga comando do automatico
	LIGA_DS_AUTO := FALSE;	
ELSE
//============================================================================
// comandos automatico
//============================================================================		
	
	//Liga dosador 
	IF  AL_GERAL = FALSE THEN
		LIGA_DS_AUTO :=TRUE;
	ELSE
		LIGA_DS_AUTO := FALSE;
	END_IF
	
	//zera velocidade do ph com peso maximo
	IF LEITURA_PESO_FLUI2 >= PRST_PESO_MAX_FLUID2 THEN
		ESPERA_FLUIDIZADOR_BAIXAR_PESO := TRUE;
	END_IF
	
	//ativa velocidade do ph com peso minimo
	IF LEITURA_PESO_FLUI2 <= PRST_PESO_MIN_FLUID2 THEN
		ESPERA_FLUIDIZADOR_BAIXAR_PESO := FALSE;
	END_IF
	
	IF ESPERA_FLUIDIZADOR_BAIXAR_PESO = FALSE THEN
		//Calculo dosagem kg/h em manual
		PRST_VEL_DS14 := (VELOCIDADE_PH2_AUTO) * (PRST_PERC_DOSA_DS14 / 100);
	ELSE
		PRST_VEL_DS14 := 0;
	END_IF
	
	//em auto desliga comando do manual
	LIGA_DS_MANUAL := FALSE;
	
END_IF

//Liga dosador
IF (( LIGA_DS_AUTO = TRUE  OR LIGA_DS_MANUAL = TRUE) ) THEN
	LIGA_DS14 := TRUE;
ELSE
	LIGA_DS14 := FALSE;
END_IF

//============================================================================
//  escrita da velocidade
//============================================================================

//Inversão da word da variavel da GVLPH: PRST_VEL_DS14, para variavel da GVLSCHENCK: PESO_DSA14
%QW15108 := %QW13578; // Endereço 852
%QW15110 := %QW13576; // Endereço 851




//============================================================================
// comandos que independem do comando manual/auto
//============================================================================

//conta tempo de homogenização
TEMPO_DESLIGA_ZERAEVENTO(IN:=BTS_LIMPEVE_DS14,PT:=T#10S);
DESLIGA_BT_LIMPA_EVE := TEMPO_DESLIGA_ZERAEVENTO.Q ;

IF DESLIGA_BT_LIMPA_EVE = TRUE THEN
	BTS_LIMPEVE_DS14 := FALSE;
END_IF

//bits de comando ============================================================
//Os bits de escrita inicio e parada da balança é invertido, por exemplo, para ligar o bit0 = false, e para parar o bit1=false

//Bit iniciar balança
IF LIGA_DS14 = FALSE THEN
	%QX15025.0 := FALSE;    //bit de ligar dosador, false para ativar	
ELSE
	%QX15025.0 := TRUE;		//bit de ligar dosador, true desativa	
END_IF

//bit parar balança
IF LIGA_DS14 = FALSE THEN
	%QX15025.1 := TRUE;		//bit de desligar dosador, true desativar
ELSE		
	%QX15025.1 := FALSE;	//bit de desligar dosador, false ativa	
END_IF

//bit limpar eventos
IF BTS_LIMPEVE_DS14 = TRUE THEN
	%QX15025.2 := TRUE;
ELSE
	%QX15025.2 := FALSE;
END_IF

//bit liberar
%QX15025.3 := TRUE;

//bit modo Volumetrico
IF BTS_MODVOL_DS14 = TRUE THEN
	%QX15025.4 := TRUE;
ELSE
	%QX15025.4 := FALSE;
END_IF
	
//bit modo Gravimetrico
IF BTS_MODGRAV_DS14 = TRUE THEN
	%QX15025.5 := TRUE;
ELSE
	%QX15025.5 := FALSE;
END_IF

//bit reinicializar Totalizador 1
IF BTS_ZERATOTAL1_DS14 = TRUE THEN
	%QX15025.6 := TRUE;
ELSE
	%QX15025.6 := FALSE;
END_IF

//Comando do Reset dos totalizadores geral, apontamento de producao
BTS_ZERATOTAL1_DS14 := BTS_RESET_TOTAL_SCHENCK;
//Tempo desliga reset totalizador 1
TMR_RESET_TOTAL1(IN:= BTS_ZERATOTAL1_DS14, PT:= T#30S);
//desliga o reset do totalizador ao zerar 
IF TMR_RESET_TOTAL1.Q = TRUE THEN
	BTS_ZERATOTAL1_DS14 := FALSE;
	BTS_RESET_TOTAL_SCHENCK := FALSE;
END_IF

//bit reinicializar Totalizador 2
IF BTS_ZERATOTAL2_DS14 = TRUE THEN
	%QX15025.7 := TRUE;
ELSE
	%QX15025.7 := FALSE;
END_IF
//Tempo desliga reset totalizador 2
TMR_RESET_TOTAL2(IN:= BTS_ZERATOTAL2_DS14, PT:= T#30S);
//desliga o reset do totalizador ao zerar 
IF TMR_RESET_TOTAL2.Q = TRUE THEN
	BTS_ZERATOTAL2_DS14 := FALSE;
END_IF

//bit Volume Sincrono
%QX15024.0 := TRUE;

//bit corre. umidade on
%QX15024.1 := TRUE;

//bit corre. umidade off
%QX15024.2 := TRUE;

//bit acionamento med. off
%QX15024.3 := TRUE;

//bit retorno da comporta PMS
%QX15024.4 := TRUE;

//bit reservado
%QX15024.5 := TRUE;

//bit reservado
%QX15024.6 := TRUE;

//bit reservado
%QX15024.7 := TRUE;


//====================================================================================
// Leitura Valores REAL 
//====================================================================================

//Totalizador1, leitura em Kg, 
//Inversão da word da variavel da GVLSCHENCK: LEITURA_TOTALIZADOR1_DSA14, para variavel da GVLPH: TOTALIZADOR1_KG 
%QW10800 := %IW16304; // Endereço Modbus 1700
%QW10802 := %IW16302; // Endereço Modbus 1701

//Totalizador2, leitura em Kg, apenas invertidos as words
//Inversão da word da variavel da GVLSCHENCK: LEITURA_TOTALIZADOR2_DSA14, para variavel da GVLPH: TOTALIZADOR2_KG 
%QW10804 := %IW16308; // Endereço Modbus 1702
%QW10806 := %IW16306; // Endereço Modbus 1703

//Totalizador3, leitura em Tonelada, invertidos as words e dividido por 1000 
//Inversão da word da variavel da GVLSCHENCK: LEITURA_TOTALIZADOR3_DSA12, para variavel da GVLPH: TOTALIZADOR3_KG 
%QW10808 := %IW16312; // Endereço Modbus 1704
%QW10810 := %IW16310; // Endereço Modbus 1705
TOTALIZADOR3_TON_DS14 := TOTALIZADOR3_KG_DS14 / 1000;

//Velocidade atual do dosador
%QW10848 := %IW16300; // Endereço Modbus 1720
%QW10850 := %IW16298; // Endereço Modbus 1721

VELOCIDADE_REAL_DS14 := VELOCIDADE_REAL2_DS14;

END_PROGRAM

// Device/Application/DSATorre
PROGRAM DSATorre
VAR
	//Rotação das bombas de alta 
	RPM:REAL;
	//P - Volume base incorporada;
	P:REAL;
	PERCENTUAL_BASE:REAL;		
	//Ds  - densidade do slurry em %
	ds:REAL;
	//Us  - Umidade do Slurry em %
	Us:REAL;
	//Ub  - Umidade do po base em %
	Ub:REAL;
	//Velocidade do Dosador
	Q:REAL;	
	//Tempo de Homogenização em TIME
	TEMPO_DESLIGA_ZERAEVENTO:TON;
	//desliga botao limpa evento
	DESLIGA_BT_LIMPA_EVE:BOOL;
	//Liga Dosador manual
	LIGA_DS_MANUAL:BOOL;
	//Liga Dosador automatico
	LIGA_DS_AUTO:BOOL;
	//Tempo desliga reset totalizador 1
	TMR_RESET_TOTAL1:TON;
	//Tempo desliga reset totalizador 2
	TMR_RESET_TOTAL2:TON;
		//Tempo retardo para ligar dosador
	TMR_RETARDO_LIGA_DOSDOR:TON;
	//Liga dosador apos tempo de retardo
	LIGA_DOSADOR_APOS_RETARDO:BOOL;
	//Tempo retardo para mover velocidade para dosador
	TMR_RETARDO_MOVE_VEL_DOSDOR:TON;
	//Move velocidade para dosador
	MOVE_VEL_DOSADOR:BOOL;
END_VAR

//POU relacionado aos comandos e alarmes do Dosador TORRE	MECHATRON DEA-D1
//Formula
//  Se Baseia no calculo de Q considerando as variaveis:
//    - vazão do po base que esta sendo soprado
//    - percental de slfato que se deseja incorporar base
//
//  Q = P*(%base) / % Sulfato
//  
//   P - Volume base incorporada;
//   %base - fraçao de base desejada
//   %sulfato - fraçao sulfato desejado na mistura
//
//    Passo 1:    calculo % base
//					% Base = %Sulfato - 100%
//				
//    Passo 2:     calculo P
//                            P:= ((RPM/11,2)*0,965 * ds * (1 - Us))/ (1 -  Ub)
//
//     RPM - rotacao motor da bomba de alta
//     Ds  - densidade do slurry em gr/l
//     Us  - Umidade do Slurry em %
//     Ub  - Umidade do po base em %
//
//     Passo3: calculo Q
//                             Q = P*PRST_RELACAO_PO_BASE / 100
//  
// multiplicar por 60 no final, pois a velocidade esta em rpm 


//Calculo da velocidade =====================================================

//se apenas bomba de alta 1 ligada
IF SD_BA1 = TRUE AND SD_BA2 = FALSE THEN
	RPM := LEITURA_VEL_ALT1;
ELSIF SD_BA2 = TRUE AND SD_BA1 = FALSE THEN    //se apenas bomba de alta 2 ligada
	RPM := LEITURA_VEL_ALT2;
ELSIF SD_BA2 = TRUE AND SD_BA1 = TRUE THEN
	RPM := LEITURA_VEL_ALT1 + LEITURA_VEL_ALT2;   // se as duas estiverem ligadas
ELSE                //quando nenhuma ligada
	RPM := 0;
END_IF


//calculo P

//Passo 1: 
//            % Base = %Sulfato - 100%

PERCENTUAL_BASE := 100 - PRST_PERC_SULFATO_DSTORRE;


//Passo 2:
//     RPM - rotacao motor da bomba de alta
//     Ds  - densidade do slurry em %
//     Us  - Umidade do Slurry em %
//     Ub  - Umidade do po base em %

ds := PRST_DS_DSTORRE/1000 ; 
Us := PRST_US_DSTORRE/100 ;
Ub := PRST_UB_DSTORRE/100 ;

 P := (((RPM/11.2)*0.965 * ds * (1 - Us))/ (1 -  Ub))*60;

 //Copia informação do P para Supervisório
 LEITURA_BASE_SOP_TORRE := P;
 
 //Passo 3:
//Calculo Q

Q := P*PRST_RELACAO_PO_BASE / 100;


//Retardo para mover velocidade dosador
TMR_RETARDO_MOVE_VEL_DOSDOR(IN:= SD_VLR, PT:= T#10S);
//move velocidade
MOVE_VEL_DOSADOR := TMR_RETARDO_MOVE_VEL_DOSDOR.Q;


//Se não estiver soprando zera velocidade do dosador
IF MOVE_VEL_DOSADOR = TRUE THEN
	PRST_VEL_DSTORRE := Q;
ELSE
	PRST_VEL_DSTORRE := 0;
END_IF



//Liga dosador manualmente ================================
IF BTS_DSTORRE = TRUE AND AL_GERAL = FALSE THEN
	IF LIGA_DS_MANUAL = TRUE THEN
		LIGA_DS_MANUAL := FALSE;
	ELSE
		LIGA_DS_MANUAL :=TRUE;
	END_IF
	BTS_DSTORRE := FALSE;
END_IF
//desliga em caso de alarme
IF AL_GERAL = TRUE THEN
	LIGA_DS_MANUAL := FALSE;
END_IF
//informa que dosador esta habilitado
IF LIGA_DS_MANUAL THEN
	DSATORRE_HAB := TRUE;
ELSE
	DSATORRE_HAB := FALSE;
END_IF

//liga se valvula retorno para torre e sopro com PH	==========================
IF SD_VLR = TRUE AND SOPRO_SEM_PH = FALSE AND AL_GERAL = FALSE THEN	
	LIGA_DS_AUTO :=TRUE;
ELSE
	LIGA_DS_AUTO := FALSE;
END_IF	
		

//Liga dosador
IF LIGA_DS_AUTO = TRUE AND LIGA_DS_MANUAL = TRUE AND AL_GERAL = FALSE  THEN
	LIGA_DSTORRE := TRUE;
ELSE
	LIGA_DSTORRE := FALSE;
END_IF


//Retardo para ligar dosador
TMR_RETARDO_LIGA_DOSDOR(IN:= LIGA_DSTORRE, PT:= T#10S);
//liga dosador
LIGA_DOSADOR_APOS_RETARDO := TMR_RETARDO_LIGA_DOSDOR.Q;

//============================================================================
//  escrita da velocidade
//============================================================================

//Inversão da word da variavel da GVLPH: PRST_VEL_DSTORRE, para variavel da GVLSCHENCK: PESO_DSATORRE
%QW15104 := %QW12768;
%QW15106 := %QW12766;

//============================================================================
// comandos que independem do comando manual/auto
//============================================================================


//bits de comando ============================================================
//Os bits de escrita inicio e parada da balança é invertido, por exemplo, para ligar o bit0 = false, e para parar o bit1=false

//Bit iniciar balança
IF LIGA_DOSADOR_APOS_RETARDO = FALSE THEN
	%QX15023.0 := FALSE;    //bit de ligar dosador, false para ativar	
ELSE
	%QX15023.0 := TRUE;		//bit de ligar dosador, true desativa	
END_IF

//bit parar balança
IF LIGA_DOSADOR_APOS_RETARDO = FALSE THEN
	%QX15023.1 := TRUE;		//bit de desligar dosador, true desativar
ELSE		
	%QX15023.1 := FALSE;	//bit de desligar dosador, false ativa	
END_IF

//bit limpar eventos
IF BTS_LIMPEVE_DSTORRE = TRUE THEN
	%QX15023.2 := TRUE;
ELSE
	%QX15023.2 := FALSE;
END_IF
//===============================RESET LIMPA EVENTOS======================

TEMPO_DESLIGA_ZERAEVENTO(IN:=BTS_LIMPEVE_DSTORRE,PT:=T#3S);
DESLIGA_BT_LIMPA_EVE := TEMPO_DESLIGA_ZERAEVENTO.Q ;

IF DESLIGA_BT_LIMPA_EVE = TRUE THEN
	BTS_LIMPEVE_DSTORRE := FALSE;
END_IF

//===============================RESET LIMPA EVENTOS======================

//bit liberar
%QX15023.3 := TRUE;

//bit modo Volumetrico
IF BTS_MODVOL_DSTORRE = TRUE THEN
	%QX15023.4 := TRUE;
ELSE
	%QX15023.4 := FALSE;
END_IF
	
//bit modo Gravimetrico
IF BTS_MODGRAV_DSTORRE = TRUE THEN
	%QX15023.5 := TRUE;
ELSE
	%QX15023.5 := FALSE;
END_IF

//bit reinicializar Totalizador 1
IF BTS_ZERATOTAL1_DSTORRE = TRUE THEN
	%QX15023.6 := TRUE;
ELSE
	%QX15023.6 := FALSE;
END_IF

//Comando do Reset dos totalizadores geral, apontamento de producao
BTS_ZERATOTAL1_DSTORRE := BTS_RESET_TOTAL_SCHENCK;
//Tempo desliga reset totalizador 1
TMR_RESET_TOTAL1(IN:= BTS_ZERATOTAL1_DSTORRE, PT:= T#15S);
//desliga o reset do totalizador ao zerar 
IF TMR_RESET_TOTAL1.Q = TRUE THEN
	BTS_ZERATOTAL1_DSTORRE := FALSE;
	BTS_RESET_TOTAL_SCHENCK := FALSE;
END_IF

//bit reinicializar Totalizador 2
IF BTS_ZERATOTAL2_DSTORRE = TRUE THEN
	%QX15023.7 := TRUE;
ELSE
	%QX15023.7 := FALSE;
END_IF
//Tempo desliga reset totalizador 2
TMR_RESET_TOTAL2(IN:= BTS_ZERATOTAL2_DSTORRE, PT:= T#15S);
//desliga o reset do totalizador ao zerar 
IF TMR_RESET_TOTAL2.Q = TRUE THEN
	BTS_ZERATOTAL2_DSTORRE := FALSE;
END_IF

//bit Volume Sincrono
%QX15022.0 := TRUE;

//bit corre. umidade on
%QX15022.1 := TRUE;

//bit corre. umidade off
%QX15022.2 := TRUE;

//bit acionamento med. off
%QX15022.3 := TRUE;

//bit retorno da comporta PMS
%QX15022.4 := TRUE;

//bit reservado
%QX15022.5 := TRUE;

//bit reservado
%QX15022.6 := TRUE;

//bit reservado
%QX15022.7 := TRUE;



//====================================================================================
// Leitura Valores REAL 
//====================================================================================

//Totalizador1, leitura em Kg, 
//Inversão da word da variavel da GVLSCHENCK: LEITURA_TOTALIZADOR1_DSATORRE, para variavel da GVLPH: TOTALIZADOR1_KG 
%QW10176 := %IW15176;
%QW10178 := %IW15174;

//Totalizador2, leitura em Kg, apenas invertidos as words
//Inversão da word da variavel da GVLSCHENCK: LEITURA_TOTALIZADOR2_DSATORRE, para variavel da GVLPH: TOTALIZADOR2_KG 
%QW10180 := %IW15236;
%QW10182 := %IW15234;

//Totalizador3, leitura em Tonelada, invertidos as words e dividido por 1000 
//Inversão da word da variavel da GVLSCHENCK: LEITURA_TOTALIZADOR3_DSATORRE, para variavel da GVLPH: TOTALIZADOR3_KG 
%QW10184 := %IW15346;
%QW10186 := %IW15344;
TOTALIZADOR3_TON_DSTORRE := TOTALIZADOR3_KG_DSTORRE / 1000;

//Velocidade atual do dosador
%QW10344 := %IW15296;
%QW10346 := %IW15294;

VELOCIDADE_REAL_DSTORRE := VELOCIDADE_REAL2_DSTORRE ;

END_PROGRAM

// Device/Application/ProdL1
PROGRAM ProdL1
VAR
	//PRODUÇÃO LINHAS ENVASE
	
//=========================	
PULSO_CNT_L1_1T: R_TRIG;
PULSO_CNT_L1_2T: R_TRIG;
PULSO_CNT_L1_3T: R_TRIG;
	CNT_PRD_L1: INT;
	//CNT_L1: BOOL;
//=========================	
	Result : RTC_STATUS;
	DATEANDTIME : EXTENDED_DATE_AND_TIME;
	xEnable : BOOL;
//=========================		
	dia: INT;
	mes: INT;
	ano: INT;
	hora: INT;
	minuto: INT;
	segundo: INT;
	
	
	
	//HoraInicio1Turno: INT;
	//MinInicio1Turno: INT;
	HoraFim1Turno: INT;
	MinFim1Turno: INT;
	//HoraInicio2Turno: INT;
	//MinInicio2Turno: INT;
	HoraFim2Turno: INT;
	MinFim2Turno: INT;
	//HoraInicio3Turno: INT;
	//MinInicio3Turno: INT;
	HoraFim3Turno: INT;
	MinFim3Turno: INT;
	EficienciaL1: INT;
	
	
	HabContL1_1T: BOOL;
	HabContL1_2T: BOOL;
	HabContL1_3T: BOOL;
	
	CNT_PRD_L1_2T: INT;
	CNT_PRD_L1_3T: INT;
	EficienciaL1_1T: REAL;
	EficienciaL1_2T: REAL;
	EficienciaL1_3T: REAL;
	
	MinDispL1_1T: REAL;
	
	ProdL1_1T_realtime: REAL;
	MinDispL1_2T: REAL;
	ProdL1_2T_realtime: REAL;
	EficL1_2T_realtime: REAL;
	MinDispL1_3T: REAL;
	ProdL1_3T_realtime: REAL;
	EficL1_3T_realtime: REAL;
	
	//TMR_SIMUL_CNT1: TON;
	//LIBERA_TMR_SIMUL: BOOL;
	EficL1_2T_projetada: REAL;
	//TMR_SIMUL_CNT2: TON;
	//LIBERA_TMR_SIMUL2T: BOOL;
	//TMR_SIMUL_CNT3: TON;
	//LIBERA_TMR_SIMUL3T: BOOL;
	EficL1_3T_projetada: REAL;
//	EficL1_1T_realtime: REAL;
	HabTemParadaL1: BOOL;
	TempParadaL1: Ton;
	horaParadaL1: INT;
	MinParadaL1: INT;
	RegistraHora: BOOL;
	Borda_des_RegistraHora: F_TRIG;
	HoraRetornoParadaL1: INT;
	MinRetornoParadaL1: INT;
	TempoParadaL1: INT;
	TotalMinParado: TON;
	HabTotalMinParado: BOOL;
	//TempoProduzindo: REAL;
	//MinDispTurnoAtual: REAL;

	refeicao: BOOL;
	DDS: BOOL;
	SETUP: BOOL;
	L1semprogramacao: BOOL;
	
END_VAR


//LÓGICA PARA ANÁLISES DE PRODUTIVADADE DA L1 DE CARTUCHOS
	dia := BYTE_TO_INT (DATEANDTIME.byDayOfMonth);
	mes := BYTE_TO_INT (DATEANDTIME.byMonth);
	ano := WORD_TO_INT (DATEANDTIME.wYear);
	hora := BYTE_TO_INT (DATEANDTIME.byHours);
	minuto := BYTE_TO_INT (DATEANDTIME.byMinutes);
	segundo := BYTE_TO_INT (DATEANDTIME.bySeconds);
	xEnable := TRUE;
	
	//HABILITA RTC==========================
	IF xEnable = TRUE THEN
	Result := GetDateAndTime(DATEANDTIME);
	END_IF
//HABILITA RTC==========================

//=====================1º TURNO ========================
	
		//HoraInicio1Turno: INT;
	
	HoraFim1Turno:= HoraInicio2Turno;
	MinFim1Turno:= MinInicio2Turno;
	HoraFim2Turno:= HoraInicio3Turno;
	MinFim2Turno:= MinInicio3Turno;
	
	//10 minutos - Reunião / DSS / Treinamento
	//20 minutosPartida de linha / Parada de Linha xxxxxxxxxx
	//15 minutosRefeições (Café / Almoço / Janta)xxxxxxxxxxxx
	//60 minutosRefeições (Café / Almoço / Janta)
	//10 minutosPartida de linha / Parada de Linha xxxxxxxxxxxxxx
			
	MinDispL1_1T := (((INT_TO_REAL (HoraFim1Turno) - INT_TO_REAL(HoraInicio1Turno) )*60)-
		INT_TO_REAL(MinInicio1Turno)+INT_TO_REAL(MinFim1Turno)-60-10);
		
			IF TempoProduzindo < 1 THEN
			TempoProduzindo :=0;
		END_IF
	
		//LÓGICA PARA VERIFICAR SE EXISTE ATRASO DE PRODUÇÃO NO INSTANTE ATUAL
		
	IF  CXS_ATRASOL1 >= 0AND HabContL1_1T = TRUE THEN 
	CXS_ATRASOL1:= REAL_TO_INT(ProdL1_1T_realtime)-CNT_PRD_L1_1T;
	END_IF
	IF  CXS_ATRASOL1 >= 0 AND HabContL1_2T = TRUE THEN 
	CXS_ATRASOL1:= REAL_TO_INT(ProdL1_2T_realtime)-CNT_PRD_L1_1T;
	END_IF
	IF  CXS_ATRASOL1 >= 0 AND HabContL1_3T = TRUE THEN 
	CXS_ATRASOL1:=REAL_TO_INT(ProdL1_2T_realtime)-CNT_PRD_L1_1T;
	END_IF
		IF  CXS_ATRASOL1  < 0 THEN 
		CXS_ATRASOL1:= 0;
		END_IF
	
	//LÓGICA PARA VERIFICAR SE EXISTE ATRASO DE PRODUÇÃO NO INSTANTE ATUAL
		
		//LÓGICA PARA CONTAR TEMPO DE PARADA
		TempParadaL1(IN:=HabTemParadaL1 ,PT:= T#30S);
		IF TempParadaL1.Q   THEN
		TotalMinParado(IN:=HabTotalMinParado ,PT:= T#1M);
		IF TotalMinParado.Q = TRUE THEN
			TempoParada := TempoParada+1;
			HabTotalMinParado := FALSE;
			ELSE
				HabTotalMinParado := TRUE;
			END_IF
		END_IF
		
		IF PULSO_CNT_L1_1T.Q = FALSE AND PULSO_CNT_L1_2T.Q = FALSE AND PULSO_CNT_L1_3T.Q = FALSE  THEN
		HabTemParadaL1 := TRUE;
		
		ELSE 	
		HabTemParadaL1 := FALSE;
		END_IF
		//LÓGICA PARA CONTAR TEMPO DE PARADA
//==============Habilita contadores 1º turno ================
IF (hora = HoraInicio1Turno AND minuto = MinInicio1Turno)  THEN
HabContL1_1T := TRUE;
HabContL1_3T := FALSE;
HabContL1_2T := FALSE;
CNT_PRD_L1_3T := 0;
CNT_PRD_L1_2T := 0;
CNT_PRD_L1_1T := 0;
TempoProduzindo :=0;
EficL1_1T_projetada:=0;
EficL1_1T_realtime :=0;
ProdL1_1T_realtime :=0;
TempoParada :=0;
CXS_ATRASOL1:=0;
END_IF 


//==============Contador e Eficiencia L1 1 TURNO de cartuchos==========
IF HabContL1_1T = TRUE THEN 
PULSO_CNT_L1_1T(CLK:=CNT_L1);
//TMR_SIMUL_CNT1(IN:=LIBERA_TMR_SIMUL ,PT:=T#9S);	
		IF PULSO_CNT_L1_1T.Q = TRUE THEN
		CNT_PRD_L1_1T := CNT_PRD_L1_1T+1;
		//LIBERA_TMR_SIMUL := FALSE;
		RegistraHora := FALSE;
		MinDispTurnoAtual := MinDispL1_1T;
//ELSE 	
	//LIBERA_TMR_SIMUL:= TRUE;
		END_IF
		
			IF hora > 5 AND hora < 11 THEN

		ProdL1_1T_realtime := (INT_TO_REAL(ProducaoProgramada_L1_1T) / (MinDispL1_1T)) * ((
		(INT_TO_REAL(hora)-INT_TO_REAL(HoraInicio1Turno))*60)-INT_TO_REAL(MinInicio1Turno) + INT_TO_REAL(minuto));
		
		TempoProduzindo :=  ((hora-HoraInicio1Turno)*60)-MinInicio1Turno+ minuto-TempoParada;
		
		EficL1_1T_realtime := ( INT_TO_REAL(CNT_PRD_L1_1T) / ProdL1_1T_realtime ) * 100 * (EficL1_1T_projetada/100);
		EficL1_1T_projetada := (ProdL1_1T_realtime / ProducaoProgramada_L1_1T) * 100;
		END_IF
		
			IF hora > 11 AND hora < 15 THEN

		ProdL1_1T_realtime := (INT_TO_REAL(ProducaoProgramada_L1_1T) / (MinDispL1_1T)) * ((
		(INT_TO_REAL(hora)-INT_TO_REAL(HoraInicio1Turno))*60)-INT_TO_REAL(MinInicio1Turno) + INT_TO_REAL(minuto)-10-60);
		
		TempoProduzindo :=  ((hora-HoraInicio1Turno)*60)-MinInicio1Turno+ minuto-TempoParada;
		
		EficL1_1T_realtime := ( INT_TO_REAL(CNT_PRD_L1_1T) / ProdL1_1T_realtime ) * 100 * (EficL1_1T_projetada/100);
		EficL1_1T_projetada := (ProdL1_1T_realtime / ProducaoProgramada_L1_1T) * 100;
		END_IF
	
END_IF
EficienciaL1_1T := (INT_TO_REAL(CNT_PRD_L1_1T) / INT_TO_REAL(ProducaoProgramada_L1_1T) ) * 100;


//=====================1º TURNO ========================

//=====================2º TURNO ========================

	//10 minutos - Reunião / DSS / Treinamento
	//20 minutosPartida de linha / Parada de Linha
	//15 minutosRefeições (Café / Almoço / Janta)
	//60 minutosRefeições (Café / Almoço / Janta)
	//10 minutosPartida de linha / Parada de Linha
	IF hora = 0 THEN 
		hora := 24;
	END_IF
	
		MinDispL1_2T := (((INT_TO_REAL (HoraFim2Turno) - INT_TO_REAL(HoraInicio2Turno) )*60)-
		INT_TO_REAL(MinInicio2Turno)+INT_TO_REAL(MinFim2Turno)-60-10);
	
//==============Contador e Eficiencia L1 2 TURNO de cartuchos==========
//==============Habilita contadores 2º turno ================
IF (hora = HoraInicio2Turno AND minuto = MinInicio2Turno)  THEN
HabContL1_2T := TRUE;
HabContL1_1T := FALSE;
CNT_PRD_L1_3T := 0;
CNT_PRD_L1_2T := 0;
CNT_PRD_L1_1T := 0;
TempoParada :=0;
TempoProduzindo :=0;
EficL1_1T_projetada:=0;
EficL1_1T_realtime :=0;
ProdL1_1T_realtime :=0;
TempoParada :=0;
CXS_ATRASOL1:=0;
END_IF 
IF HabContL1_2T = TRUE THEN 
PULSO_CNT_L1_2T(CLK:=CNT_L1);
//TMR_SIMUL_CNT2(IN:=LIBERA_TMR_SIMUL2T ,PT:=T#7S);
		IF PULSO_CNT_L1_2T.Q = TRUE  THEN
		CNT_PRD_L1_2T := CNT_PRD_L1_2T+1;
		//LIBERA_TMR_SIMUL2T := FALSE;
		MinDispTurnoAtual := MinDispL1_2T;
//ELSE 	
	//LIBERA_TMR_SIMUL2T:= TRUE;	
		END_IF
		CNT_PRD_L1_1T := CNT_PRD_L1_2T ;
		EficL1_1T_projetada:=EficL1_2T_projetada;
		EficL1_1T_realtime :=EficL1_2T_realtime;
		ProdL1_1T_realtime :=ProdL1_1T_realtime;
		
			IF hora > 13 AND hora < 19 THEN

		ProdL1_2T_realtime := (INT_TO_REAL(ProducaoProgramada_L1_2T) / (MinDispL1_2T)) * ((
		(INT_TO_REAL(hora)-INT_TO_REAL(HoraInicio2Turno))*60)-INT_TO_REAL(MinInicio2Turno) + INT_TO_REAL(minuto));
		
		TempoProduzindo :=  ((hora-HoraInicio2Turno)*60)-MinInicio2Turno+ minuto-TempoParada;
		
		EficL1_2T_realtime := ( INT_TO_REAL(CNT_PRD_L1_2T) / ProdL1_2T_realtime ) * 100 * (EficL1_2T_projetada/100);
		EficL1_2T_projetada := (ProdL1_2T_realtime / ProducaoProgramada_L1_2T) * 100;
		END_IF
		IF hora > 19 AND hora < 23 THEN

		ProdL1_2T_realtime := (INT_TO_REAL(ProducaoProgramada_L1_2T) / (MinDispL1_2T)) * ((
		(INT_TO_REAL(hora)-INT_TO_REAL(HoraInicio2Turno))*60)-INT_TO_REAL(MinInicio2Turno) + INT_TO_REAL(minuto)-10-60);
		
		TempoProduzindo :=  ((hora-HoraInicio2Turno)*60)-MinInicio2Turno+ minuto-TempoParada;
		
		EficL1_2T_realtime := ( INT_TO_REAL(CNT_PRD_L1_2T) / ProdL1_2T_realtime ) * 100 * (EficL1_2T_projetada/100);
		EficL1_2T_projetada := (ProdL1_2T_realtime / ProducaoProgramada_L1_2T) * 100;
		END_IF
END_IF
EficienciaL1_2T := (INT_TO_REAL (CNT_PRD_L1_2T) / INT_TO_REAL (ProducaoProgramada_L1_2T)  ) * 100;

//=====================2º TURNO ========================

//=====================3º TURNO ========================
//==============Contador e Eficiencia L1 3 TURNO de cartuchos==========

//==============Habilita contadores 3º turno ================
//10 minutos - Reunião / DSS / Treinamento
	//20 minutosPartida de linha / Parada de Linha
	//15 minutosRefeições (Café / Almoço / Janta)
	//60 minutosRefeições (Café / Almoço / Janta)
	//10 minutosPartida de linha / Parada de Linha
	IF hora = 0 THEN 
		hora := 24;
	END_IF
	
		MinDispL1_3T := (((INT_TO_REAL (HoraFim3Turno) - INT_TO_REAL(HoraInicio3Turno) )*60)-
		INT_TO_REAL(MinInicio3Turno)+INT_TO_REAL(MinFim3Turno)-60-10);
		
	
//==============Contador e Eficiencia L1 3 TURNO de cartuchos==========
//==============Habilita contadores 3º turno ================
IF (hora = HoraInicio3Turno AND minuto = MinInicio3Turno)  THEN
HabContL1_3T := TRUE;
HabContL1_2T := FALSE;
HabContL1_1T := FALSE;
CNT_PRD_L1_3T := 0;
CNT_PRD_L1_2T := 0;
CNT_PRD_L1_1T := 0;
TempoParada :=0;
TempoProduzindo :=0;
EficL1_1T_projetada:=0;
EficL1_1T_realtime :=0;
ProdL1_1T_realtime :=0;
TempoParada :=0;
CXS_ATRASOL1:=0;
END_IF 

IF HabContL1_3T = TRUE THEN 
PULSO_CNT_L1_3T(CLK:=CNT_L1);	
		IF PULSO_CNT_L1_3T.Q = TRUE THEN
		CNT_PRD_L1_3T := CNT_PRD_L1_3T+1;	
			CNT_PRD_L1_1T := CNT_PRD_L1_3T ;
		EficL1_1T_projetada:=EficL1_3T_projetada;
		EficL1_1T_realtime :=EficL1_3T_realtime;
		ProdL1_1T_realtime :=ProdL1_3T_realtime;
		END_IF
		IF hora > 21 AND hora <= 24 THEN

		ProdL1_3T_realtime := (INT_TO_REAL(ProducaoProgramada_L1_3T) / (MinDispL1_3T)) * ((
		(INT_TO_REAL(hora)-INT_TO_REAL(HoraInicio3Turno))*60)-INT_TO_REAL(MinInicio3Turno) + INT_TO_REAL(minuto));
		
		TempoProduzindo :=  ((hora-HoraInicio3Turno)*60)-MinInicio3Turno+ minuto-TempoParada;
	
		EficL1_3T_realtime := ( INT_TO_REAL(CNT_PRD_L1_3T) / ProdL1_3T_realtime ) * 100 *(EficL1_3T_projetada/100) ;
		EficL1_3T_projetada := (ProdL1_3T_realtime / ProducaoProgramada_L1_3T) * 100;
		END_IF
		IF ((hora > 0 ) AND minuto > 30) AND hora < 2 THEN

		ProdL1_3T_realtime := (INT_TO_REAL(ProducaoProgramada_L1_3T) / (MinDispL1_3T)) * ((
		(INT_TO_REAL(hora)-INT_TO_REAL(HoraInicio3Turno))*60)-INT_TO_REAL(MinInicio3Turno) + INT_TO_REAL(minuto)-10-60);
		
		TempoProduzindo :=  ((hora-HoraInicio3Turno)*60)-MinInicio3Turno+ minuto-TempoParada;
	
		EficL1_3T_realtime := ( INT_TO_REAL(CNT_PRD_L1_3T) / ProdL1_3T_realtime ) * 100 *(EficL1_3T_projetada/100) ;
		EficL1_3T_projetada := (ProdL1_3T_realtime / ProducaoProgramada_L1_3T) * 100;
		END_IF
END_IF


EficienciaL1_3T := (INT_TO_REAL (CNT_PRD_L1_3T) / INT_TO_REAL (ProducaoProgramada_L1_3T)  ) * 100;


IF (hora = HoraInicio3Turno AND minuto = MinInicio3Turno)  THEN
HabContL1_3T := TRUE;
HabContL1_2T := FALSE;
END_IF 

IF HabContL1_3T = TRUE THEN 
PULSO_CNT_L1_3T(CLK:=CNT_L1);
//TMR_SIMUL_CNT3(IN:=LIBERA_TMR_SIMUL3T ,PT:=T#8S);
		IF PULSO_CNT_L1_3T.Q = TRUE  THEN
		CNT_PRD_L1_3T := CNT_PRD_L1_3T+1;
		//LIBERA_TMR_SIMUL3T := FALSE;
		MinDispTurnoAtual := MinDispL1_3T;
//ELSE 	
	//LIBERA_TMR_SIMUL3T:= TRUE;	
		END_IF
		END_IF
	
	
EficienciaL1_3T := (INT_TO_REAL (CNT_PRD_L1_3T) / INT_TO_REAL(ProducaoProgramada_L1_3T)  ) * 100;
//=====================3º TURNO ========================

IF (hora = 11 AND minuto = 0) OR (hora = 19 AND minuto = 0) OR (hora = 1 AND minuto = 30)  THEN
	refeicao := TRUE;
	END_IF
	IF (hora = 11 AND minuto = 40) OR  (hora = 20 AND minuto = 0)  OR  (hora = 2 AND minuto = 30)  THEN
	refeicao := FALSE;
	END_IF 
	
	IF (hora = 6 AND minuto = 0) OR (hora = 20 AND minuto = 0) OR (hora = 2 AND minuto = 30)  THEN
	DDS := TRUE;
	END_IF
	IF (hora = 6 AND minuto = 10) OR  (hora = 20 AND minuto = 10)  OR  (hora = 2 AND minuto = 40)  THEN
	DDS := FALSE;
	END_IF 
	IF (hora = 6 AND minuto = 0) OR (hora = 14 AND minuto = 20) OR (hora = 22 AND minuto = 30)  THEN
	SETUP := TRUE;
	END_IF
	IF (hora = 6 AND minuto = 30) OR  (hora = 14 AND minuto = 50)  OR  (hora = 23 AND minuto = 0)  THEN
	SETUP := FALSE;
	END_IF 
	
//STATUS DA LINHA 1
//STATUS DO EQUIPAMENTO
//0- SEM PROGRAMAÇÃO
//1- PRODUZINDO
//2- PARADA
//3- REFEIÇÃO
//4- DDS
//5- SETUP

IF ProducaoProgramada_L1_1T = 0 AND HabContL1_1T = TRUE AND TempParadaL1.Q = TRUE  THEN
	Status_L1 := 0;
	L1semprogramacao :=TRUE;
	END_IF
		IF ProducaoProgramada_L1_1T > 0 AND HabContL1_1T = TRUE THEN 
		L1semprogramacao :=FALSE;
		END_IF
	
IF ProducaoProgramada_L1_2T = 0 AND HabContL1_2T = TRUE  AND TempParadaL1.Q = TRUE THEN
	Status_L1 := 0;
	L1semprogramacao :=TRUE;
		END_IF
			IF ProducaoProgramada_L1_2T > 0 AND HabContL1_2T = TRUE THEN 
				L1semprogramacao :=FALSE;
				END_IF
				
IF ProducaoProgramada_L1_3T = 0 AND HabContL1_3T = TRUE AND TempParadaL1.Q = TRUE THEN
	Status_L1 := 0;
	L1semprogramacao :=TRUE;
		END_IF
			IF ProducaoProgramada_L1_3T > 0 AND HabContL1_3T = TRUE THEN 
			L1semprogramacao :=FALSE;
			END_IF
	
IF TempParadaL1.Q = FALSE THEN
	Status_L1 := 1;
END_IF

	IF refeicao = FALSE AND SETUP = FALSE AND DDS = FALSE AND TempParadaL1.Q = TRUE AND L1semprogramacao = FALSE THEN
	Status_L1 := 2;
	END_IF

IF refeicao = TRUE AND TempParadaL1.Q = TRUE THEN
Status_L1 := 3;
END_IF

IF DDS = TRUE AND TempParadaL1.Q = TRUE THEN
Status_L1 := 4;
END_IF

//IF SETUP = TRUE THEN
//Status_L1 := 5;
//END_IF


//STATUS DA LINHA 1

END_PROGRAM

// Device/Application/ProdL2
PROGRAM ProdL2
VAR
	//PRODUÇÃO LINHAS ENVASE
	
//=========================	
PULSO_CNT_L2_1T: R_TRIG;
PULSO_CNT_L2_2T: R_TRIG;
PULSO_CNT_L2_3T: R_TRIG;
	CNT_PRD_L2: INT;
	//CNT_L2: BOOL;
//=========================	
	Result : RTC_STATUS;
	DATEANDTIME : EXTENDED_DATE_AND_TIME;
	xEnable : BOOL;
//=========================		
	dia: INT;
	mes: INT;
	ano: INT;
	hora: INT;
	minuto: INT;
	segundo: INT;
	
	
	
	//HoraInicio1Turno: INT;
	//MinInicio1Turno: INT;
	HoraFim1Turno: INT;
	MinFim1Turno: INT;
	//HoraInicio2Turno: INT;
	//MinInicio2Turno: INT;
	HoraFim2Turno: INT;
	MinFim2Turno: INT;
	//HoraInicio3Turno: INT;
	//MinInicio3Turno: INT;
	HoraFim3Turno: INT;
	MinFim3Turno: INT;
	EficienciaL2: INT;
	
	
	HabContL2_1T: BOOL;
	HabContL2_2T: BOOL;
	HabContL2_3T: BOOL;
	
	CNT_PRD_L2_2T: INT;
	CNT_PRD_L2_3T: INT;
	EficienciaL2_1T: REAL;
	EficienciaL2_2T: REAL;
	EficienciaL2_3T: REAL;
	
	MinDispL2_1T: REAL;
	
	ProdL2_1T_realtime: REAL;
	MinDispL2_2T: REAL;
	ProdL2_2T_realtime: REAL;
	EficL2_2T_realtime: REAL;
	MinDispL2_3T: REAL;
	ProdL2_3T_realtime: REAL;
	EficL2_3T_realtime: REAL;
	
	//TMR_SIMUL_CNT1: TON;
	//LIBERA_TMR_SIMUL: BOOL;
	EficL2_2T_projetada: REAL;
	//TMR_SIMUL_CNT2: TON;
	//LIBERA_TMR_SIMUL2T: BOOL;
	//TMR_SIMUL_CNT3: TON;
	//LIBERA_TMR_SIMUL3T: BOOL;
	EficL2_3T_projetada: REAL;
//	EficL2_1T_realtime: REAL;
	HabTemParadaL2: BOOL;
	TempParadaL2: Ton;
	horaParadaL2: INT;
	MinParadaL2: INT;
	RegistraHora: BOOL;
	Borda_des_RegistraHora: F_TRIG;
	HoraRetornoParadaL2: INT;
	MinRetornoParadaL2: INT;
	TempoParadaL2L2: INT;
	TotalMinParado: TON;
	HabTotalMinParado: BOOL;
	//TempoProduzindoL2: REAL;
	//MinDispTurnoAtual: REAL;

	refeicao: BOOL;
	DDS: BOOL;
	SETUP: BOOL;
	L2semprogramacao: BOOL;
END_VAR


//LÓGICA PARA ANÁLISES DE PRODUTIVADADE DA L2 DE CARTUCHOS
	dia := BYTE_TO_INT (DATEANDTIME.byDayOfMonth);
	mes := BYTE_TO_INT (DATEANDTIME.byMonth);
	ano := WORD_TO_INT (DATEANDTIME.wYear);
	hora := BYTE_TO_INT (DATEANDTIME.byHours);
	minuto := BYTE_TO_INT (DATEANDTIME.byMinutes);
	segundo := BYTE_TO_INT (DATEANDTIME.bySeconds);
	xEnable := TRUE;
	
	//HABILITA RTC==========================
	IF xEnable = TRUE THEN
	Result := GetDateAndTime(DATEANDTIME);
	END_IF
//HABILITA RTC==========================

//=====================1º TURNO ========================
	
		//HoraInicio1Turno: INT;
	
	HoraFim1Turno:= HoraInicio2Turno;
	MinFim1Turno:= MinInicio2Turno;
	HoraFim2Turno:= HoraInicio3Turno;
	MinFim2Turno:= MinInicio3Turno;
	
	//10 minutos - Reunião / DSS / Treinamento
	//20 minutosPartida de linha / Parada de Linha xxxxxxxxxx
	//15 minutosRefeições (Café / Almoço / Janta)xxxxxxxxxxxx
	//60 minutosRefeições (Café / Almoço / Janta)
	//10 minutosPartida de linha / Parada de Linha xxxxxxxxxxxxxx
			
	MinDispL2_1T := (((INT_TO_REAL (HoraFim1Turno) - INT_TO_REAL(HoraInicio1Turno) )*60)-
		INT_TO_REAL(MinInicio1Turno)+INT_TO_REAL(MinFim1Turno)-60-10);
		
			IF TempoProduzindoL2 < 1 THEN
			TempoProduzindoL2 :=0;
			END_IF
	
	//LÓGICA PARA VERIFICAR SE EXISTE ATRASO DE PRODUÇÃO NO INSTANTE ATUAL
		
	IF  CXS_ATRASOL2 >= 0 AND HabContL2_1T = TRUE THEN 
	CXS_ATRASOL2:= REAL_TO_INT(ProdL2_1T_realtime)-CNT_PRD_L2_1T;
		END_IF
	IF  CXS_ATRASOL2 >= 0 AND HabContL2_2T = TRUE THEN 
	CXS_ATRASOL2:= REAL_TO_INT(ProdL2_2T_realtime)-CNT_PRD_L2_1T;
	END_IF
	IF  CXS_ATRASOL2 >= 0 AND HabContL2_3T = TRUE THEN 
	CXS_ATRASOL2:=REAL_TO_INT(ProdL2_2T_realtime)-CNT_PRD_L2_1T;
	END_IF
		IF  CXS_ATRASOL2  < 0 THEN 
	CXS_ATRASOL2:= 0;
		END_IF
	
	//LÓGICA PARA VERIFICAR SE EXISTE ATRASO DE PRODUÇÃO NO INSTANTE ATUAL	
		
		//LÓGICA PARA CONTAR TEMPO DE PARADA
		TempParadaL2(IN:=HabTemParadaL2 ,PT:= T#30S);
		IF TempParadaL2.Q   THEN
		TotalMinParado(IN:=HabTotalMinParado ,PT:= T#1M);
		IF TotalMinParado.Q = TRUE THEN
			TempoParadaL2 := TempoParadaL2+1;
			HabTotalMinParado := FALSE;
			ELSE
				HabTotalMinParado := TRUE;
			END_IF
		END_IF
		
		IF PULSO_CNT_L2_1T.Q = FALSE AND PULSO_CNT_L2_2T.Q = FALSE AND PULSO_CNT_L2_3T.Q = FALSE  THEN
		HabTemParadaL2 := TRUE;
		
		ELSE 	
		HabTemParadaL2 := FALSE;
		END_IF
		//LÓGICA PARA CONTAR TEMPO DE PARADA
//==============Habilita contadores 1º turno ================
IF (hora = HoraInicio1Turno AND minuto = MinInicio1Turno)  THEN
HabContL2_1T := TRUE;
HabContL2_3T := FALSE;
HabContL2_2T := FALSE;
CNT_PRD_L2_3T := 0;
CNT_PRD_L2_2T := 0;
CNT_PRD_L2_1T := 0;
TempoProduzindoL2 :=0;
EficL2_1T_projetada:=0;
EficL2_1T_realtime :=0;
ProdL2_1T_realtime :=0;
TempoParadaL2 :=0;
CXS_ATRASOL2:=0;
END_IF 


//==============Contador e Eficiencia L2 1 TURNO de cartuchos==========
IF HabContL2_1T = TRUE THEN 
PULSO_CNT_L2_1T(CLK:=CNT_L2);
//TMR_SIMUL_CNT1(IN:=LIBERA_TMR_SIMUL ,PT:=T#9S);	
		IF PULSO_CNT_L2_1T.Q = TRUE THEN
		CNT_PRD_L2_1T := CNT_PRD_L2_1T+1;
		//LIBERA_TMR_SIMUL := FALSE;
		RegistraHora := FALSE;
		MinDispTurnoAtual := MinDispL2_1T;
//ELSE 	
	//LIBERA_TMR_SIMUL:= TRUE;
		END_IF
		
			IF hora > 5 AND hora < 11 THEN

		ProdL2_1T_realtime := (INT_TO_REAL(ProducaoProgramada_L2_1T) / (MinDispL2_1T)) * ((
		(INT_TO_REAL(hora)-INT_TO_REAL(HoraInicio1Turno))*60)-INT_TO_REAL(MinInicio1Turno) + INT_TO_REAL(minuto));
		
		TempoProduzindoL2 :=  ((hora-HoraInicio1Turno)*60)-MinInicio1Turno+ minuto-TempoParadaL2;
		
		EficL2_1T_realtime := ( INT_TO_REAL(CNT_PRD_L2_1T) / ProdL2_1T_realtime ) * 100 * (EficL2_1T_projetada/100);
		EficL2_1T_projetada := (ProdL2_1T_realtime / ProducaoProgramada_L2_1T) * 100;
		END_IF
		
			IF hora > 11 AND hora < 15 THEN

		ProdL2_1T_realtime := (INT_TO_REAL(ProducaoProgramada_L2_1T) / (MinDispL2_1T)) * ((
		(INT_TO_REAL(hora)-INT_TO_REAL(HoraInicio1Turno))*60)-INT_TO_REAL(MinInicio1Turno) + INT_TO_REAL(minuto)-10-60);
		
		TempoProduzindoL2 :=  ((hora-HoraInicio1Turno)*60)-MinInicio1Turno+ minuto-TempoParadaL2;
		
		EficL2_1T_realtime := ( INT_TO_REAL(CNT_PRD_L2_1T) / ProdL2_1T_realtime ) * 100 * (EficL2_1T_projetada/100);
		EficL2_1T_projetada := (ProdL2_1T_realtime / ProducaoProgramada_L2_1T) * 100;
		END_IF
	
END_IF
EficienciaL2_1T := (INT_TO_REAL(CNT_PRD_L2_1T) / INT_TO_REAL(ProducaoProgramada_L2_1T) ) * 100;


//=====================1º TURNO ========================

//=====================2º TURNO ========================

	//10 minutos - Reunião / DSS / Treinamento
	//20 minutosPartida de linha / Parada de Linha
	//15 minutosRefeições (Café / Almoço / Janta)
	//60 minutosRefeições (Café / Almoço / Janta)
	//10 minutosPartida de linha / Parada de Linha
	IF hora = 0 THEN 
		hora := 24;
	END_IF
	
		MinDispL2_2T := (((INT_TO_REAL (HoraFim2Turno) - INT_TO_REAL(HoraInicio2Turno) )*60)-
		INT_TO_REAL(MinInicio2Turno)+INT_TO_REAL(MinFim2Turno)-60-10);
	
//==============Contador e Eficiencia L2 2 TURNO de cartuchos==========
//==============Habilita contadores 2º turno ================
IF (hora = HoraInicio2Turno AND minuto = MinInicio2Turno)  THEN
HabContL2_2T := TRUE;
HabContL2_1T := FALSE;
CNT_PRD_L2_3T := 0;
CNT_PRD_L2_2T := 0;
CNT_PRD_L2_1T := 0;
TempoParadaL2 :=0;
TempoProduzindoL2 :=0;
EficL2_1T_projetada:=0;
EficL2_1T_realtime :=0;
ProdL2_1T_realtime :=0;
TempoParadaL2 :=0;
CXS_ATRASOL2:=0;
END_IF 
IF HabContL2_2T = TRUE THEN 
PULSO_CNT_L2_2T(CLK:=CNT_L2);
//TMR_SIMUL_CNT2(IN:=LIBERA_TMR_SIMUL2T ,PT:=T#7S);
		IF PULSO_CNT_L2_2T.Q = TRUE  THEN
		CNT_PRD_L2_2T := CNT_PRD_L2_2T+1;
		//LIBERA_TMR_SIMUL2T := FALSE;
		MinDispTurnoAtual := MinDispL2_2T;
//ELSE 	
	//LIBERA_TMR_SIMUL2T:= TRUE;	
		END_IF
		CNT_PRD_L2_1T := CNT_PRD_L2_2T ;
		EficL2_1T_projetada:=EficL2_2T_projetada;
		EficL2_1T_realtime :=EficL2_2T_realtime;
		ProdL2_1T_realtime :=ProdL2_1T_realtime;
		
			IF hora > 13 AND hora < 19 THEN

		ProdL2_2T_realtime := (INT_TO_REAL(ProducaoProgramada_L2_2T) / (MinDispL2_2T)) * ((
		(INT_TO_REAL(hora)-INT_TO_REAL(HoraInicio2Turno))*60)-INT_TO_REAL(MinInicio2Turno) + INT_TO_REAL(minuto));
		
		TempoProduzindoL2 :=  ((hora-HoraInicio2Turno)*60)-MinInicio2Turno+ minuto-TempoParadaL2;
		
		EficL2_2T_realtime := ( INT_TO_REAL(CNT_PRD_L2_2T) / ProdL2_2T_realtime ) * 100 * (EficL2_2T_projetada/100);
		EficL2_2T_projetada := (ProdL2_2T_realtime / ProducaoProgramada_L2_2T) * 100;
		END_IF
		IF hora > 19 AND hora < 23 THEN

		ProdL2_2T_realtime := (INT_TO_REAL(ProducaoProgramada_L2_2T) / (MinDispL2_2T)) * ((
		(INT_TO_REAL(hora)-INT_TO_REAL(HoraInicio2Turno))*60)-INT_TO_REAL(MinInicio2Turno) + INT_TO_REAL(minuto)-10-60);
		
		TempoProduzindoL2 :=  ((hora-HoraInicio2Turno)*60)-MinInicio2Turno+ minuto-TempoParadaL2;
		
		EficL2_2T_realtime := ( INT_TO_REAL(CNT_PRD_L2_2T) / ProdL2_2T_realtime ) * 100 * (EficL2_2T_projetada/100);
		EficL2_2T_projetada := (ProdL2_2T_realtime / ProducaoProgramada_L2_2T) * 100;
		END_IF
END_IF
EficienciaL2_2T := (INT_TO_REAL (CNT_PRD_L2_2T) / INT_TO_REAL (ProducaoProgramada_L2_2T)  ) * 100;

//=====================2º TURNO ========================

//=====================3º TURNO ========================
//==============Contador e Eficiencia L2 3 TURNO de cartuchos==========

//==============Habilita contadores 3º turno ================
//10 minutos - Reunião / DSS / Treinamento
	//20 minutosPartida de linha / Parada de Linha
	//15 minutosRefeições (Café / Almoço / Janta)
	//60 minutosRefeições (Café / Almoço / Janta)
	//10 minutosPartida de linha / Parada de Linha
	IF hora = 0 THEN 
		hora := 24;
	END_IF
	
		MinDispL2_3T := (((INT_TO_REAL (HoraFim3Turno) - INT_TO_REAL(HoraInicio3Turno) )*60)-
		INT_TO_REAL(MinInicio3Turno)+INT_TO_REAL(MinFim3Turno)-60-10);
		
	
//==============Contador e Eficiencia L2 3 TURNO de cartuchos==========
//==============Habilita contadores 3º turno ================
IF (hora = HoraInicio3Turno AND minuto = MinInicio3Turno)  THEN
HabContL2_3T := TRUE;
HabContL2_2T := FALSE;
HabContL2_1T := FALSE;
CNT_PRD_L2_3T := 0;
CNT_PRD_L2_2T := 0;
CNT_PRD_L2_1T := 0;
TempoParadaL2 :=0;
TempoProduzindoL2 :=0;
EficL2_1T_projetada:=0;
EficL2_1T_realtime :=0;
ProdL2_1T_realtime :=0;
TempoParadaL2 :=0;
CXS_ATRASOL1:=0;
END_IF 

IF HabContL2_3T = TRUE THEN 
PULSO_CNT_L2_3T(CLK:=CNT_L2);	
		IF PULSO_CNT_L2_3T.Q = TRUE THEN
		CNT_PRD_L2_3T := CNT_PRD_L2_3T+1;	
			CNT_PRD_L2_1T := CNT_PRD_L2_3T ;
		EficL2_1T_projetada:=EficL2_3T_projetada;
		EficL2_1T_realtime :=EficL2_3T_realtime;
		ProdL2_1T_realtime :=ProdL2_3T_realtime;
		END_IF
		IF hora > 21 AND hora <= 24 THEN

		ProdL2_3T_realtime := (INT_TO_REAL(ProducaoProgramada_L2_3T) / (MinDispL2_3T)) * ((
		(INT_TO_REAL(hora)-INT_TO_REAL(HoraInicio3Turno))*60)-INT_TO_REAL(MinInicio3Turno) + INT_TO_REAL(minuto));
		
		TempoProduzindoL2 :=  ((hora-HoraInicio3Turno)*60)-MinInicio3Turno+ minuto-TempoParadaL2;
	
		EficL2_3T_realtime := ( INT_TO_REAL(CNT_PRD_L2_3T) / ProdL2_3T_realtime ) * 100 *(EficL2_3T_projetada/100) ;
		EficL2_3T_projetada := (ProdL2_3T_realtime / ProducaoProgramada_L2_3T) * 100;
		END_IF
		IF ((hora > 0 ) AND minuto > 30) AND hora < 2 THEN

		ProdL2_3T_realtime := (INT_TO_REAL(ProducaoProgramada_L2_3T) / (MinDispL2_3T)) * ((
		(INT_TO_REAL(hora)-INT_TO_REAL(HoraInicio3Turno))*60)-INT_TO_REAL(MinInicio3Turno) + INT_TO_REAL(minuto)-10-60);
		
		TempoProduzindoL2 :=  ((hora-HoraInicio3Turno)*60)-MinInicio3Turno+ minuto-TempoParadaL2;
	
		EficL2_3T_realtime := ( INT_TO_REAL(CNT_PRD_L2_3T) / ProdL2_3T_realtime ) * 100 *(EficL2_3T_projetada/100) ;
		EficL2_3T_projetada := (ProdL2_3T_realtime / ProducaoProgramada_L2_3T) * 100;
		END_IF
END_IF


EficienciaL2_3T := (INT_TO_REAL (CNT_PRD_L2_3T) / INT_TO_REAL (ProducaoProgramada_L2_3T)  ) * 100;


IF (hora = HoraInicio3Turno AND minuto = MinInicio3Turno)  THEN
HabContL2_3T := TRUE;
HabContL2_2T := FALSE;
END_IF 

IF HabContL2_3T = TRUE THEN 
PULSO_CNT_L2_3T(CLK:=CNT_L2);
//TMR_SIMUL_CNT3(IN:=LIBERA_TMR_SIMUL3T ,PT:=T#8S);
		IF PULSO_CNT_L2_3T.Q = TRUE  THEN
		CNT_PRD_L2_3T := CNT_PRD_L2_3T+1;
		//LIBERA_TMR_SIMUL3T := FALSE;
		MinDispTurnoAtual := MinDispL2_3T;
//ELSE 	
	//LIBERA_TMR_SIMUL3T:= TRUE;	
		END_IF
		END_IF
	
	
EficienciaL2_3T := (INT_TO_REAL (CNT_PRD_L2_3T) / INT_TO_REAL(ProducaoProgramada_L2_3T)  ) * 100;
//=====================3º TURNO ========================

IF (hora = 11 AND minuto = 0) OR (hora = 19 AND minuto = 0) OR (hora = 1 AND minuto = 30)  THEN
	refeicao := TRUE;
	END_IF
	IF (hora = 11 AND minuto = 40) OR  (hora = 20 AND minuto = 0)  OR  (hora = 2 AND minuto = 30)  THEN
	refeicao := FALSE;
	END_IF 
	
	IF (hora = 6 AND minuto = 0) OR (hora = 20 AND minuto = 0) OR (hora = 2 AND minuto = 30)  THEN
	DDS := TRUE;
	END_IF
	IF (hora = 6 AND minuto = 10) OR  (hora = 20 AND minuto = 10)  OR  (hora = 2 AND minuto = 40)  THEN
	DDS := FALSE;
	END_IF 
	IF (hora = 6 AND minuto = 0) OR (hora = 14 AND minuto = 20) OR (hora = 22 AND minuto = 30)  THEN
	SETUP := TRUE;
	END_IF
	IF (hora = 6 AND minuto = 30) OR  (hora = 14 AND minuto = 50)  OR  (hora = 23 AND minuto = 0)  THEN
	SETUP := FALSE;
	END_IF 
	
//STATUS DA LINHA 2
//STATUS DO EQUIPAMENTO
//0- SEM PROGRAMAÇÃO
//1- PRODUZINDO
//2- PARADA
//3- REFEIÇÃO
//4- DDS
//5- SETUP

IF ProducaoProgramada_L2_1T = 0 AND HabContL2_1T = TRUE AND TempParadaL2.Q = TRUE THEN
	Status_L2 := 0;
	L2semprogramacao :=TRUE;
	END_IF
		IF ProducaoProgramada_L2_1T > 0 AND HabContL2_1T = TRUE THEN 
		L2semprogramacao :=FALSE;
		END_IF
	
IF ProducaoProgramada_L2_2T = 0 AND HabContL2_2T = TRUE AND TempParadaL2.Q = TRUE THEN
	Status_L2 := 0;
	L2semprogramacao :=TRUE;
		END_IF
			IF ProducaoProgramada_L2_2T > 0 AND HabContL2_2T = TRUE THEN 
				L2semprogramacao :=FALSE;
				END_IF
				
IF ProducaoProgramada_L2_3T = 0 AND HabContL2_3T = TRUE AND TempParadaL2.Q = TRUE THEN
	Status_L2 := 0;
	L2semprogramacao :=TRUE;
		END_IF
			IF ProducaoProgramada_L2_3T > 0 AND HabContL2_3T = TRUE THEN 
			L2semprogramacao :=FALSE;
			END_IF
	
IF TempParadaL2.Q = FALSE  THEN
	Status_L2 := 1;
END_IF

	IF refeicao = FALSE AND SETUP = FALSE AND DDS = FALSE AND TempParadaL2.Q = TRUE AND L2semprogramacao = FALSE THEN
	Status_L2 := 2;
	END_IF

IF refeicao = TRUE  AND TempParadaL2.Q = TRUE THEN
Status_L2 := 3;
END_IF

IF DDS = TRUE AND TempParadaL2.Q = TRUE THEN
Status_L2 := 4;
END_IF

//IF SETUP = TRUE THEN
//Status_L2 := 5;
//END_IF
//STATUS DA LINHA 2

END_PROGRAM

// Device/Application/ProdL3
PROGRAM ProdL3
VAR
	//PRODUÇÃO LINHAS ENVASE
	
//=========================	
PULSO_CNT_L3_1T: R_TRIG;
PULSO_CNT_L3_2T: R_TRIG;
PULSO_CNT_L3_3T: R_TRIG;
	CNT_PRD_L3: INT;
	//CNT_L3: BOOL;
//=========================	
	Result : RTC_STATUS;
	DATEANDTIME : EXTENDED_DATE_AND_TIME;
	xEnable : BOOL;
//=========================		
	dia: INT;
	mes: INT;
	ano: INT;
	hora: INT;
	minuto: INT;
	segundo: INT;
	
	
	
	//HoraInicio1Turno: INT;
	//MinInicio1Turno: INT;
	HoraFim1Turno: INT;
	MinFim1Turno: INT;
	//HoraInicio2Turno: INT;
	//MinInicio2Turno: INT;
	HoraFim2Turno: INT;
	MinFim2Turno: INT;
	//HoraInicio3Turno: INT;
	//MinInicio3Turno: INT;
	HoraFim3Turno: INT;
	MinFim3Turno: INT;
	EficienciaL3: INT;
	
	
	HabContL3_1T: BOOL;
	HabContL3_2T: BOOL;
	HabContL3_3T: BOOL;
	
	CNT_PRD_L3_2T: INT;
	CNT_PRD_L3_3T: INT;
	EficienciaL3_1T: REAL;
	EficienciaL3_2T: REAL;
	EficienciaL3_3T: REAL;
	
	MinDispL3_1T: REAL;
	
	ProdL3_1T_realtime: REAL;
	MinDispL3_2T: REAL;
	ProdL3_2T_realtime: REAL;
	EficL3_2T_realtime: REAL;
	MinDispL3_3T: REAL;
	ProdL3_3T_realtime: REAL;
	EficL3_3T_realtime: REAL;
	
	//TMR_SIMUL_CNT1: TON;
	//LIBERA_TMR_SIMUL: BOOL;
	EficL3_2T_projetada: REAL;
	//TMR_SIMUL_CNT2: TON;
	//LIBERA_TMR_SIMUL3T: BOOL;
	//TMR_SIMUL_CNT3: TON;
	//LIBERA_TMR_SIMUL3T: BOOL;
	EficL3_3T_projetada: REAL;
//	EficL3_1T_realtime: REAL;
	HabTemParadaL3: BOOL;
	TempParadaL3: Ton;
	horaParadaL3: INT;
	MinParadaL3: INT;
	RegistraHora: BOOL;
	Borda_des_RegistraHora: F_TRIG;
	HoraRetornoParadaL3: INT;
	MinRetornoParadaL3: INT;
	TempoParadaL3L3: INT;
	TotalMinParado: TON;
	HabTotalMinParado: BOOL;
	//TempoProduzindoL3: REAL;
	//MinDispTurnoAtual: REAL;

	refeicao: BOOL;
	DDS: BOOL;
	SETUP: BOOL;
	L3semprogramacao: BOOL;
	AuxProdL3: BOOL;
END_VAR


//LÓGICA PARA ANÁLISES DE PRODUTIVADADE DA L3 DE CARTUCHOS
	dia := BYTE_TO_INT (DATEANDTIME.byDayOfMonth);
	mes := BYTE_TO_INT (DATEANDTIME.byMonth);
	ano := WORD_TO_INT (DATEANDTIME.wYear);
	hora := BYTE_TO_INT (DATEANDTIME.byHours);
	minuto := BYTE_TO_INT (DATEANDTIME.byMinutes);
	segundo := BYTE_TO_INT (DATEANDTIME.bySeconds);
	xEnable := TRUE;
	
	//HABILITA RTC==========================
	IF xEnable = TRUE THEN
	Result := GetDateAndTime(DATEANDTIME);
	END_IF
//HABILITA RTC==========================

//=====================1º TURNO ========================
	
		//HoraInicio1Turno: INT;
	
	HoraFim1Turno:= HoraInicio2Turno;
	MinFim1Turno:= MinInicio2Turno;
	HoraFim2Turno:= HoraInicio3Turno;
	MinFim2Turno:= MinInicio3Turno;
	
	//10 minutos - Reunião / DSS / Treinamento
	//20 minutosPartida de linha / Parada de Linha xxxxxxxxxx
	//15 minutosRefeições (Café / Almoço / Janta)xxxxxxxxxxxx
	//60 minutosRefeições (Café / Almoço / Janta)
	//10 minutosPartida de linha / Parada de Linha xxxxxxxxxxxxxx
			
	MinDispL3_1T := (((INT_TO_REAL (HoraFim1Turno) - INT_TO_REAL(HoraInicio1Turno) )*60)-
		INT_TO_REAL(MinInicio1Turno)+INT_TO_REAL(MinFim1Turno)-60-10);
		
		IF TempoProduzindoL3 < 1 THEN
			TempoProduzindoL3 :=0;
		END_IF
	
	//LÓGICA PARA VERIFICAR SE EXISTE ATRASO DE PRODUÇÃO NO INSTANTE ATUAL
		
	IF  CXS_ATRASOL3 >= 0 AND HabContL3_1T = TRUE THEN 
	CXS_ATRASOL3:= REAL_TO_INT(ProdL3_1T_realtime)-CNT_PRD_L3_1T;
	END_IF
	IF  CXS_ATRASOL3 >= 0 AND HabContL3_2T = TRUE THEN 
	CXS_ATRASOL3:= REAL_TO_INT(ProdL3_2T_realtime)-CNT_PRD_L3_1T;
	END_IF
	IF  CXS_ATRASOL3 >= 0 AND HabContL3_3T = TRUE THEN 
	CXS_ATRASOL3:=REAL_TO_INT(ProdL3_2T_realtime)-CNT_PRD_L3_1T;
	END_IF
		IF  CXS_ATRASOL3  < 0 THEN 
		CXS_ATRASOL3:= 0;
		END_IF
	
	
	//LÓGICA PARA VERIFICAR SE EXISTE ATRASO DE PRODUÇÃO NO INSTANTE ATUAL		
		//LÓGICA PARA CONTAR TEMPO DE PARADA
		TempParadaL3(IN:=HabTemParadaL3 ,PT:= T#30S);
		IF TempParadaL3.Q   THEN
		TotalMinParado(IN:=HabTotalMinParado ,PT:= T#1M);
		IF TotalMinParado.Q = TRUE THEN
			TempoParadaL3 := TempoParadaL3+1;
			HabTotalMinParado := FALSE;
			ELSE
				HabTotalMinParado := TRUE;
			END_IF
		END_IF
		
		IF PULSO_CNT_L3_1T.Q = FALSE AND PULSO_CNT_L3_2T.Q = FALSE AND PULSO_CNT_L3_3T.Q = FALSE  THEN
		HabTemParadaL3 := TRUE;
		
		ELSE 	
		HabTemParadaL3 := FALSE;
		END_IF
		//LÓGICA PARA CONTAR TEMPO DE PARADA
//==============Habilita contadores 1º turno ================
IF (hora = HoraInicio1Turno AND minuto = MinInicio1Turno)  THEN
HabContL3_1T := TRUE;
HabContL3_3T := FALSE;
HabContL3_2T := FALSE;
CNT_PRD_L3_3T := 0;
CNT_PRD_L3_2T := 0;
CNT_PRD_L3_1T := 0;
TempoProduzindoL3 :=0;
EficL3_1T_projetada:=0;
EficL3_1T_realtime :=0;
ProdL3_1T_realtime :=0;
TempoParadaL3 :=0;
CXS_ATRASOL3:=0;
END_IF 


//==============Contador e Eficiencia L3 1 TURNO de cartuchos==========
IF HabContL3_1T = TRUE THEN 
PULSO_CNT_L3_1T(CLK:=CNT_L3);
//TMR_SIMUL_CNT1(IN:=LIBERA_TMR_SIMUL ,PT:=T#9S);	
		IF PULSO_CNT_L3_1T.Q = TRUE THEN
		CNT_PRD_L3_1T := CNT_PRD_L3_1T+1;
		//LIBERA_TMR_SIMUL := FALSE;
		RegistraHora := FALSE;
		MinDispTurnoAtual := MinDispL3_1T;
//ELSE 	
	//LIBERA_TMR_SIMUL:= TRUE;
		END_IF
		
			IF hora > 5 AND hora < 11 THEN

		ProdL3_1T_realtime := (INT_TO_REAL(ProducaoProgramada_L3_1T) / (MinDispL3_1T)) * ((
		(INT_TO_REAL(hora)-INT_TO_REAL(HoraInicio1Turno))*60)-INT_TO_REAL(MinInicio1Turno) + INT_TO_REAL(minuto));
		
		TempoProduzindoL3 :=  ((hora-HoraInicio1Turno)*60)-MinInicio1Turno+ minuto-TempoParadaL3;
		
		EficL3_1T_realtime := ( INT_TO_REAL(CNT_PRD_L3_1T) / ProdL3_1T_realtime ) * 100 * (EficL3_1T_projetada/100);
		EficL3_1T_projetada := (ProdL3_1T_realtime / ProducaoProgramada_L3_1T) * 100;
		END_IF
		
			IF hora > 11 AND hora < 15 THEN

		ProdL3_1T_realtime := (INT_TO_REAL(ProducaoProgramada_L3_1T) / (MinDispL3_1T)) * ((
		(INT_TO_REAL(hora)-INT_TO_REAL(HoraInicio1Turno))*60)-INT_TO_REAL(MinInicio1Turno) + INT_TO_REAL(minuto)-10-60);
		
		TempoProduzindoL3 :=  ((hora-HoraInicio1Turno)*60)-MinInicio1Turno+ minuto-TempoParadaL3;
		
		EficL3_1T_realtime := ( INT_TO_REAL(CNT_PRD_L3_1T) / ProdL3_1T_realtime ) * 100 * (EficL3_1T_projetada/100);
		EficL3_1T_projetada := (ProdL3_1T_realtime / ProducaoProgramada_L3_1T) * 100;
		END_IF
	
END_IF
EficienciaL3_1T := (INT_TO_REAL(CNT_PRD_L3_1T) / INT_TO_REAL(ProducaoProgramada_L3_1T) ) * 100;


//=====================1º TURNO ========================

//=====================2º TURNO ========================

	//10 minutos - Reunião / DSS / Treinamento
	//20 minutosPartida de linha / Parada de Linha
	//15 minutosRefeições (Café / Almoço / Janta)
	//60 minutosRefeições (Café / Almoço / Janta)
	//10 minutosPartida de linha / Parada de Linha
	IF hora = 0 THEN 
		hora := 24;
	END_IF
	
		MinDispL3_2T := (((INT_TO_REAL (HoraFim2Turno) - INT_TO_REAL(HoraInicio2Turno) )*60)-
		INT_TO_REAL(MinInicio2Turno)+INT_TO_REAL(MinFim2Turno)-60-10);
	
//==============Contador e Eficiencia L3 2 TURNO de cartuchos==========
//==============Habilita contadores 2º turno ================
IF (hora = HoraInicio2Turno AND minuto = MinInicio2Turno)  THEN
HabContL3_2T := TRUE;
HabContL3_1T := FALSE;
CNT_PRD_L3_3T := 0;
CNT_PRD_L3_2T := 0;
CNT_PRD_L3_1T := 0;
TempoParadaL3 :=0;
TempoProduzindoL3 :=0;
EficL3_1T_projetada:=0;
EficL3_1T_realtime :=0;
ProdL3_1T_realtime :=0;
TempoParadaL3 :=0;
CXS_ATRASOL3:=0;
END_IF 
IF HabContL3_2T = TRUE THEN 
PULSO_CNT_L3_2T(CLK:=CNT_L3);
//TMR_SIMUL_CNT2(IN:=LIBERA_TMR_SIMUL3T ,PT:=T#7S);
		IF PULSO_CNT_L3_2T.Q = TRUE  THEN
		CNT_PRD_L3_2T := CNT_PRD_L3_2T+1;
		//LIBERA_TMR_SIMUL3T := FALSE;
		MinDispTurnoAtual := MinDispL3_2T;
//ELSE 	
	//LIBERA_TMR_SIMUL3T:= TRUE;	
		END_IF
		CNT_PRD_L3_1T := CNT_PRD_L3_2T ;
		EficL3_1T_projetada:=EficL3_2T_projetada;
		EficL3_1T_realtime :=EficL3_2T_realtime;
		ProdL3_1T_realtime :=ProdL3_1T_realtime;
		
			IF hora > 13 AND hora < 19 THEN

		ProdL3_2T_realtime := (INT_TO_REAL(ProducaoProgramada_L3_T2) / (MinDispL3_2T)) * ((
		(INT_TO_REAL(hora)-INT_TO_REAL(HoraInicio2Turno))*60)-INT_TO_REAL(MinInicio2Turno) + INT_TO_REAL(minuto));
		
		TempoProduzindoL3 :=  ((hora-HoraInicio2Turno)*60)-MinInicio2Turno+ minuto-TempoParadaL3;
		
		EficL3_2T_realtime := ( INT_TO_REAL(CNT_PRD_L3_2T) / ProdL3_2T_realtime ) * 100 * (EficL3_2T_projetada/100);
		EficL3_2T_projetada := (ProdL3_2T_realtime / ProducaoProgramada_L3_T2) * 100;
		END_IF
		IF hora > 19 AND hora < 23 THEN

		ProdL3_2T_realtime := (INT_TO_REAL(ProducaoProgramada_L3_T2) / (MinDispL3_2T)) * ((
		(INT_TO_REAL(hora)-INT_TO_REAL(HoraInicio2Turno))*60)-INT_TO_REAL(MinInicio2Turno) + INT_TO_REAL(minuto)-10-60);
		
		TempoProduzindoL3 :=  ((hora-HoraInicio2Turno)*60)-MinInicio2Turno+ minuto-TempoParadaL3;
		
		EficL3_2T_realtime := ( INT_TO_REAL(CNT_PRD_L3_2T) / ProdL3_2T_realtime ) * 100 * (EficL3_2T_projetada/100);
		EficL3_2T_projetada := (ProdL3_2T_realtime / ProducaoProgramada_L3_T2) * 100;
		END_IF
END_IF
EficienciaL3_2T := (INT_TO_REAL (CNT_PRD_L3_2T) / INT_TO_REAL (ProducaoProgramada_L3_T2)  ) * 100;

//=====================2º TURNO ========================

//=====================3º TURNO ========================
//==============Contador e Eficiencia L3 3 TURNO de cartuchos==========

//==============Habilita contadores 3º turno ================
//10 minutos - Reunião / DSS / Treinamento
	//20 minutosPartida de linha / Parada de Linha
	//15 minutosRefeições (Café / Almoço / Janta)
	//60 minutosRefeições (Café / Almoço / Janta)
	//10 minutosPartida de linha / Parada de Linha
	IF hora = 0 THEN 
		hora := 24;
	END_IF
	
		MinDispL3_3T := (((INT_TO_REAL (HoraFim3Turno) - INT_TO_REAL(HoraInicio3Turno) )*60)-
		INT_TO_REAL(MinInicio3Turno)+INT_TO_REAL(MinFim3Turno)-60-10);
		
	
//==============Contador e Eficiencia L3 3 TURNO de cartuchos==========
//==============Habilita contadores 3º turno ================
IF (hora = HoraInicio3Turno AND minuto = MinInicio3Turno)  THEN
HabContL3_3T := TRUE;
HabContL3_2T := FALSE;
HabContL3_1T := FALSE;
CNT_PRD_L3_3T := 0;
CNT_PRD_L3_2T := 0;
CNT_PRD_L3_1T := 0;
TempoParadaL3 :=0;
TempoProduzindoL3 :=0;
EficL3_1T_projetada:=0;
EficL3_1T_realtime :=0;
ProdL3_1T_realtime :=0;
TempoParadaL3 :=0;
CXS_ATRASOL1:=0;
END_IF 

IF HabContL3_3T = TRUE THEN 
PULSO_CNT_L3_3T(CLK:=CNT_L3);	
		IF PULSO_CNT_L3_3T.Q = TRUE THEN
		CNT_PRD_L3_3T := CNT_PRD_L3_3T+1;	
			CNT_PRD_L3_1T := CNT_PRD_L3_3T ;
		EficL3_1T_projetada:=EficL3_3T_projetada;
		EficL3_1T_realtime :=EficL3_3T_realtime;
		ProdL3_1T_realtime :=ProdL3_3T_realtime;
		END_IF
		IF hora > 21 AND hora <= 24 THEN

		ProdL3_3T_realtime := (INT_TO_REAL(ProducaoProgramada_L3_T3) / (MinDispL3_3T)) * ((
		(INT_TO_REAL(hora)-INT_TO_REAL(HoraInicio3Turno))*60)-INT_TO_REAL(MinInicio3Turno) + INT_TO_REAL(minuto));
		
		TempoProduzindoL3 :=  ((hora-HoraInicio3Turno)*60)-MinInicio3Turno+ minuto-TempoParadaL3;
	
		EficL3_3T_realtime := ( INT_TO_REAL(CNT_PRD_L3_3T) / ProdL3_3T_realtime ) * 100 *(EficL3_3T_projetada/100) ;
		EficL3_3T_projetada := (ProdL3_3T_realtime / ProducaoProgramada_L3_T3) * 100;
		END_IF
		IF ((hora > 0 ) AND minuto > 30) AND hora < 2 THEN

		ProdL3_3T_realtime := (INT_TO_REAL(ProducaoProgramada_L3_T3) / (MinDispL3_3T)) * ((
		(INT_TO_REAL(hora)-INT_TO_REAL(HoraInicio3Turno))*60)-INT_TO_REAL(MinInicio3Turno) + INT_TO_REAL(minuto)-10-60);
		
		TempoProduzindoL3 :=  ((hora-HoraInicio3Turno)*60)-MinInicio3Turno+ minuto-TempoParadaL3;
	
		EficL3_3T_realtime := ( INT_TO_REAL(CNT_PRD_L3_3T) / ProdL3_3T_realtime ) * 100 *(EficL3_3T_projetada/100) ;
		EficL3_3T_projetada := (ProdL3_3T_realtime / ProducaoProgramada_L3_T3) * 100;
		END_IF
END_IF


EficienciaL3_3T := (INT_TO_REAL (CNT_PRD_L3_3T) / INT_TO_REAL (ProducaoProgramada_L3_T3)  ) * 100;


IF (hora = HoraInicio3Turno AND minuto = MinInicio3Turno)  THEN
HabContL3_3T := TRUE;
HabContL3_2T := FALSE;
END_IF 

IF HabContL3_3T = TRUE THEN 
PULSO_CNT_L3_3T(CLK:=CNT_L3);
//TMR_SIMUL_CNT3(IN:=LIBERA_TMR_SIMUL3T ,PT:=T#8S);
		IF PULSO_CNT_L3_3T.Q = TRUE  THEN
		CNT_PRD_L3_3T := CNT_PRD_L3_3T+1;
		//LIBERA_TMR_SIMUL3T := FALSE;
		MinDispTurnoAtual := MinDispL3_3T;
//ELSE 	
	//LIBERA_TMR_SIMUL3T:= TRUE;	
		END_IF
		END_IF
	
	
EficienciaL3_3T := (INT_TO_REAL (CNT_PRD_L3_3T) / INT_TO_REAL(ProducaoProgramada_L3_T3)  ) * 100;
//=====================3º TURNO ========================

IF (hora = 11 AND minuto = 0) OR (hora = 19 AND minuto = 0) OR (hora = 1 AND minuto = 30)  THEN
	refeicao := TRUE;
	END_IF
	IF (hora = 11 AND minuto = 40) OR  (hora = 20 AND minuto = 0)  OR  (hora = 2 AND minuto = 30)  THEN
	refeicao := FALSE;
	END_IF 
	
	IF (hora = 6 AND minuto = 0) OR (hora = 20 AND minuto = 0) OR (hora = 2 AND minuto = 30)  THEN
	DDS := TRUE;
	END_IF
	IF (hora = 6 AND minuto = 10) OR  (hora = 20 AND minuto = 10)  OR  (hora = 2 AND minuto = 40)  THEN
	DDS := FALSE;
	END_IF 
	IF (hora = 6 AND minuto = 0) OR (hora = 14 AND minuto = 20) OR (hora = 22 AND minuto = 30)  THEN
	SETUP := TRUE;
	END_IF
	IF (hora = 6 AND minuto = 30) OR  (hora = 14 AND minuto = 50)  OR  (hora = 23 AND minuto = 0)  THEN
	SETUP := FALSE;
	END_IF 
	
//STATUS DA LINHA 3
//STATUS DO EQUIPAMENTO
//0- SEM PROGRAMAÇÃO
//1- PRODUZINDO
//2- PARADA
//3- REFEIÇÃO
//4- DDS
//5- SETUP

IF ProducaoProgramada_L3_1T = 0 AND HabContL3_1T = TRUE AND TempParadaL3.Q = TRUE THEN
	Status_L3 := 0;
	L3semprogramacao :=TRUE;
	END_IF
		IF ProducaoProgramada_L3_1T > 0 AND HabContL3_1T = TRUE THEN 
		L3semprogramacao :=FALSE;
		END_IF
	
IF ProducaoProgramada_L3_T2 = 0 AND HabContL3_2T = TRUE AND TempParadaL3.Q = TRUE THEN
	Status_L3 := 0;
	L3semprogramacao :=TRUE;
		END_IF
			IF ProducaoProgramada_L3_T2 > 0 AND HabContL3_2T = TRUE THEN 
				L3semprogramacao :=FALSE;
				END_IF
				
IF ProducaoProgramada_L3_T3 = 0 AND HabContL3_3T = TRUE AND TempParadaL3.Q = TRUE THEN
	Status_L3 := 0;
	L3semprogramacao :=TRUE;
		END_IF
			IF ProducaoProgramada_L3_T3 > 0 AND HabContL3_3T = TRUE THEN 
			L3semprogramacao :=FALSE;
			END_IF
	
IF   TempParadaL3.Q = FALSE  THEN
	
	Status_L3 := 1; // Produzindo
END_IF

	IF refeicao = FALSE AND SETUP = FALSE AND DDS = FALSE AND TempParadaL3.Q = TRUE AND L3semprogramacao = FALSE THEN
	Status_L3 := 2; // Parada
	AuxProdL3 := TRUE;
	END_IF

	IF TempParadaL3.Q = FALSE AND AuxProdL3 = TRUE THEN
		Status_L3 := 6; // Fim da parada
		AuxProdL3 := FALSE;
	END_IF
	
IF refeicao = TRUE AND TempParadaL3.Q = TRUE THEN
Status_L3 := 3; // Refeição
END_IF

IF DDS = TRUE AND TempParadaL3.Q = TRUE THEN
Status_L3 := 4; // DDS
END_IF

//IF SETUP = TRUE THEN
//Status_L3 := 5;
//END_IF

//STATUS DA LINHA 3

END_PROGRAM

// Device/Application/ProdL4
PROGRAM ProdL4
VAR
	//PRODUÇÃO LINHAS ENVASE
	
//=========================	
PULSO_CNT_L4_1T: R_TRIG;
PULSO_CNT_L4_2T: R_TRIG;
PULSO_CNT_L4_3T: R_TRIG;
	CNT_PRD_L4: INT;
	//CNT_L4: BOOL;
//=========================	
	Result : RTC_STATUS;
	DATEANDTIME : EXTENDED_DATE_AND_TIME;
	xEnable : BOOL;
//=========================		
	dia: INT;
	mes: INT;
	ano: INT;
	hora: INT;
	minuto: INT;
	segundo: INT;
	
	
	
	//HoraInicio1Turno: INT;
	//MinInicio1Turno: INT;
	HoraFim1Turno: INT;
	MinFim1Turno: INT;
	//HoraInicio2Turno: INT;
	//MinInicio2Turno: INT;
	HoraFim2Turno: INT;
	MinFim2Turno: INT;
	//HoraInicio3Turno: INT;
	//MinInicio3Turno: INT;
	HoraFim3Turno: INT;
	MinFim3Turno: INT;
	EficienciaL4: INT;
	
	
	HabContL4_1T: BOOL;
	HabContL4_2T: BOOL;
	HabContL4_3T: BOOL;
	
	CNT_PRD_L4_2T: INT;
	CNT_PRD_L4_3T: INT;
	EficienciaL4_1T: REAL;
	EficienciaL4_2T: REAL;
	EficienciaL4_3T: REAL;
	
	MinDispL4_1T: REAL;
	
	ProdL4_1T_realtime: REAL;
	MinDispL4_2T: REAL;
	ProdL4_2T_realtime: REAL;
	EficL4_2T_realtime: REAL;
	MinDispL4_3T: REAL;
	ProdL4_3T_realtime: REAL;
	EficL4_3T_realtime: REAL;
	
	//TMR_SIMUL_CNT1: TON;
	//LIBERA_TMR_SIMUL: BOOL;
	EficL4_2T_projetada: REAL;
	//TMR_SIMUL_CNT2: TON;
	//LIBERA_TMR_SIMUL4T: BOOL;
	//TMR_SIMUL_CNT3: TON;
	//LIBERA_TMR_SIMUL4T: BOOL;
	EficL4_3T_projetada: REAL;
//	EficL4_1T_realtime: REAL;
	HabTemParadaL4: BOOL;
	TempParadaL4: Ton;
	horaParadaL4: INT;
	MinParadaL4: INT;
	RegistraHora: BOOL;
	Borda_des_RegistraHora: F_TRIG;
	HoraRetornoParadaL4: INT;
	MinRetornoParadaL4: INT;
	TempoParadaL4L4: INT;
	TotalMinParado: TON;
	HabTotalMinParado: BOOL;
	//TempoProduzindoL4: REAL;
	//MinDispTurnoAtual: REAL;

	refeicao: BOOL;
	DDS: BOOL;
	SETUP: BOOL;
END_VAR

VAR_INPUT
	L4semprogramacao: BOOL;
END_VAR


//LÓGICA PARA ANÁLISES DE PRODUTIVADADE DA L4 DE CARTUCHOS
	dia := BYTE_TO_INT (DATEANDTIME.byDayOfMonth);
	mes := BYTE_TO_INT (DATEANDTIME.byMonth);
	ano := WORD_TO_INT (DATEANDTIME.wYear);
	hora := BYTE_TO_INT (DATEANDTIME.byHours);
	minuto := BYTE_TO_INT (DATEANDTIME.byMinutes);
	segundo := BYTE_TO_INT (DATEANDTIME.bySeconds);
	xEnable := TRUE;
	
	//HABILITA RTC==========================
	IF xEnable = TRUE THEN
	Result := GetDateAndTime(DATEANDTIME);
	END_IF
//HABILITA RTC==========================

//=====================1º TURNO ========================
	
		//HoraInicio1Turno: INT;
	
	HoraFim1Turno:= HoraInicio2Turno;
	MinFim1Turno:= MinInicio2Turno;
	HoraFim2Turno:= HoraInicio3Turno;
	MinFim2Turno:= MinInicio3Turno;
	
	
	//10 minutos - Reunião / DSS / Treinamento
	//20 minutosPartida de linha / Parada de Linha xxxxxxxxxx
	//15 minutosRefeições (Café / Almoço / Janta)xxxxxxxxxxxx
	//60 minutosRefeições (Café / Almoço / Janta)
	//10 minutosPartida de linha / Parada de Linha xxxxxxxxxxxxxx
			
	MinDispL4_1T := (((INT_TO_REAL (HoraFim1Turno) - INT_TO_REAL(HoraInicio1Turno) )*60)-
		INT_TO_REAL(MinInicio1Turno)+INT_TO_REAL(MinFim1Turno)-60-10);
		
		IF TempoProduzindoL4 < 1 THEN
			TempoProduzindoL4 :=0;
		END_IF
	
			//LÓGICA PARA VERIFICAR SE EXISTE ATRASO DE PRODUÇÃO NO INSTANTE ATUAL
		
	IF  CXS_ATRASOL4 >= 0 AND HabContL4_1T = TRUE THEN 
	CXS_ATRASOL4:= REAL_TO_INT(ProdL4_1T_realtime)-CNT_PRD_L4_1T;
	END_IF
	IF  CXS_ATRASOL4 >= 0 AND HabContL4_2T = TRUE THEN 
	CXS_ATRASOL4:= REAL_TO_INT(ProdL4_2T_realtime)-CNT_PRD_L4_1T;
	END_IF
	IF  CXS_ATRASOL4 >= 0 AND HabContL4_3T = TRUE THEN 
	CXS_ATRASOL4:=REAL_TO_INT(ProdL4_2T_realtime)-CNT_PRD_L4_1T;
	END_IF
		IF  CXS_ATRASOL4  < 0 THEN 
		CXS_ATRASOL4:= 0;
		END_IF
	
	
	//LÓGICA PARA VERIFICAR SE EXISTE ATRASO DE PRODUÇÃO NO INSTANTE ATUAL
		
		//LÓGICA PARA CONTAR TEMPO DE PARADA
		TempParadaL4(IN:=HabTemParadaL4 ,PT:= T#30S);
		IF TempParadaL4.Q   THEN
		TotalMinParado(IN:=HabTotalMinParado ,PT:= T#1M);
		IF TotalMinParado.Q = TRUE THEN
			TempoParadaL4 := TempoParadaL4+1;
			HabTotalMinParado := FALSE;
			ELSE
				HabTotalMinParado := TRUE;
			END_IF
		END_IF
		
